// ---- P2POUs/BasicFunction/10_MES/CS_CodeTcp.TcPOU
FUNCTION_BLOCK PUBLIC CS_CodeTcp
VAR_INPUT
	bLON                           :BOOL; 	//  扫码开
	sRemoteHost: T_IPv4Addr; 			//扫码枪IP地址;
	bComOpen                  :BOOL; 	 //扫码Tcp 开
	binit_tcp:BOOL;							//功能块初始化，所有状态全部清零；
END_VAR

VAR_OUTPUT
	bComOpenDone          :BOOL;  //扫码Tcp 打开OK
    bCodeConError             :BOOL;//扫码通讯故障
	bDone                         :BOOL; //扫码完成
    bCodeError                  :BOOL;//扫码故障	
    strCode                       :STRING;//条码结果
	Code_State:INT;						//扫码结果 1：OK  2：NG
END_VAR

VAR_IN_OUT

END_VAR

VAR
	bLOFF                          :BOOL; 	//扫码关	
	bComClose                  :BOOL;  	//扫码Tcp 关
	fbTcpCon:FB_SocketConnect;
	fbTcpSend:FB_SocketSend;
	fbTcpRec:FB_SocketReceive;
	fbTcpClose: FB_SocketClose;
	bConnect: BOOL;//打开TCP连接;
	bClose: BOOL;		//关闭TCP连接;
	hTcpSock: T_HSOCKET;
	StrSend:STRING;
	StrReceive:STRING;
	StrReceive2:STRING:='';//clean;
	fbUdpCreate:FB_SocketUdpCreate;
	hUdp: T_HSOCKET;
	bCreate: BOOL;
	port: UDINT:=23;
	bSendTcp: BOOL;
	bReceiveTcp: BOOL;
	fbSwingHalt2: MC_Halt;
    TON01:TON;
	Lenth: UINT;
	StrSend2: STRING;
	bSendTcp2: BOOL;
	iComSetp: INT;
	bRectiveEN: BOOL;
	TON_3: Ton;
	TON_4: TON;
	tTon5: BOOL;
	TON_5: TON;
END_VAR




	Config();
	
	M_SendReceive();


	
	

	
	
	
	

	
	
	
	
	
	
	
	
	
	
	
	
	
	
	
	
	
(*	
   fbUdpCreate(
	sSrvNetId:= , 
	sLocalHost:= , 
	nLocalPort:= port, 
	bExecute:=bCreate , 
	tTimeout:= , 
	bBusy=> , 
	bError=> , 
	nErrId=> , 
	hSocket=> hUdp);
	
	
	*)

ACTION Config:
(*
功能块初始化；
外部给一个上升沿;
*)
TON_3(IN:=binit_tcp , PT:=T#2MS , Q=> , ET=> ); 
IF binit_tcp THEN
	iComSetp:=0;
	bComOpenDone:=FALSE;
    bCodeConError:=FALSE;
	bCodeError:=FALSE;
	bConnect:=FALSE;
	bClose :=TRUE;
	bDone:=FALSE;
    strCode:=StrReceive2;	 
	StrReceive:=StrReceive2;	 
	Code_State:=0;
	bRectiveEN:=FALSE;
	bSendTcp:=FALSE;
END_IF
IF TON_3.Q THEN
	binit_tcp:=FALSE;
	bClose :=FALSE;
END_IF

(*************************************************************)

IF bComOpen THEN
    bComOpenDone:=FALSE;
    bCodeConError:=FALSE;
    iComSetp:=100;
END_IF
  
 IF bComClose THEN
     bComOpenDone:=FALSE;
     bCodeConError:=FALSE;
     iComSetp:=200;
END_IF 
  

 CASE iComSetp OF 
   100:
	   bConnect:=TRUE;	
	   bClose:=FALSE;
	   bComOpen:=FALSE;
	   iComSetp:=110;
  110:
	  IF bConnect  THEN
		  bConnect:=FALSE;	
		   iComSetp:=120;
	  ELSIF fbTcpCon.bError THEN
		  iComSetp:=999;
	 END_IF
  120:
	 IF fbTcpCon.hSocket.handle>0  THEN
		bComOpenDone:=TRUE;//扫码枪连接成功；
		 iComSetp:=666;
	 ELSIF  NOT fbTcpCon.bBusy AND fbTcpCon.hSocket.handle=0  THEN
		iComSetp:=999;
	 END_IF

  200:
	   bConnect:=FALSE;	
	   bClose:=TRUE;
	   bComClose:=FALSE;
       iComSetp:=210;
  210:
	  IF fbTcpClose.bBusy THEN
		  bConnect:=FALSE;	
		   iComSetp:=666;
	 END_IF
  
  999:
	   bCodeConError:=TRUE;
	   iComSetp:=0;
END_CASE

fbTcpCon(
	sSrvNetId:= ''   ,                                     
	sRemoteHost:=sRemoteHost,     
	nRemotePort:= 23, 
	bExecute:=bConnect , 
	tTimeout:= , 
	bBusy=> , 
	bError=> , 
	nErrId=> , 
	hSocket=>hTcpSock );

fbTcpClose(
	sSrvNetId:= ''   , 
	hSocket:=hTcpSock , 
	bExecute:=bClose , 
	tTimeout:=T#5S , 
	bBusy=> , 
	bError=> , 
	nErrId=> );
END_ACTION

ACTION M_SendReceive:
(*
扫码失败返回“NG”；
 MEMSET(ADR(StrReceive2),0,SIZEOF(StrReceive2)); 
*)
TON_5(IN:=tTon5, PT:=T#4S , Q=> , ET=> ); 
IF TON_5.Q THEN
	tTon5:=FALSE;
END_IF

 IF bLON   AND  bComOpenDone   THEN
	StrReceive2:='$00$00$00$00$00$00$00$00$00$00$00$00$00$00$00$00$00$00$00$00$00$00$00$00$00$00$00$00$00$00$00$00';
	StrReceive:=StrReceive2;	 
	strCode:=StrReceive2;
	tTon5:=TRUE;
	IF StrReceive='' THEN
		 StrSend:='+';
		 bSendTcp:=TRUE;
		 bLON:=FALSE;
		 bDone:=FALSE;
		 bCodeError:=FALSE;
		 strCode:='';
		 Lenth:=SIZEOF(StrSend);
		 bRectiveEN:=TRUE;
	  END_IF
 END_IF
 

  IF bLOFF OR bCodeConError THEN
     StrSend:='+';
	 bSendTcp:=TRUE;
	 bLOFF:=FALSE;
	 bDone:=FALSE;
	 bCodeError:=FALSE;
	 strCode:='';
	 bComOpenDone:=FALSE;
	 iComSetp:=0;
	 Code_State:=0;
	 Lenth:=SIZEOF(StrSend2);
  END_IF

 //发送； 
fbTcpSend(
		sSrvNetId:= , 
		hSocket:=hTcpSock , 
		cbLen:=SIZEOF(StrSend), 
		pSrc:= ADR(StrSend), 
		bExecute:= bSendTcp, 
		tTimeout:= T#2S , 
		bBusy=> , 
		bError=> , 
		nErrId=> );
	
	IF TON01.Q THEN
		bSendTcp:=FALSE;
	END_IF

	
//接收;
bReceiveTcp:=tTon5 AND NOT bReceiveTcp AND  bRectiveEN     ;
fbTcpRec(
	sSrvNetId:= , 
	hSocket:= hTcpSock, 
	cbLen:=SIZEOF(StrReceive) , 
	pDest:=ADR(StrReceive) , 
	bExecute:=bReceiveTcp , 
	tTimeout:= T#5S, 
	bBusy=> , 
	bError=> , 
	nErrId=> , 
	nRecBytes=> );
	
(*接收数据超时；	*)

TON_4(IN:=bRectiveEN, PT:=T#4S , Q=> , ET=> ); 
IF TON_4.Q THEN
		IF(  StrReceive='' )OR ( LEN(STR:=StrReceive )<>2 AND LEN(STR:=StrReceive )<>15 )THEN	
				strCode:=StrReceive;
			   StrReceive:='';
			   bRectiveEN:=FALSE;
			   bCodeError:=TRUE;
			   Code_State:=2;			//拍照失败；
		END_IF
END_IF

(*数据位数不对报警*)
IF tTon5 AND LEN(STR:=StrReceive )<>0 AND LEN(STR:=StrReceive )<>2 AND LEN(STR:=StrReceive )<>15  THEN
				strCode:=StrReceive;
			   StrReceive:='';
			   bRectiveEN:=FALSE;
			   bCodeError:=TRUE;
			   Code_State:=2;			//拍照失败；
END_IF

(*截取数据判断；*)
IF StrReceive<>''THEN
		IF NOT bLON AND NOT fbTcpRec.bBusy THEN
			bRectiveEN:=FALSE;
			bSendTcp:=FALSE;
		END_IF

IF tTon5 AND LEN(STR:=StrReceive )>=2 AND LEN(STR:=StrReceive )<=15 AND FIND(STR1:=StrReceive , STR2:='ERROR' )=0 THEN
	  strCode:=StrReceive;
	  StrReceive:='';
     bRectiveEN:=FALSE;
	 bDone:=TRUE;
	 		IF strCode='NG' THEN
				Code_State:=2;//拍照失败；
			ELSE
				Code_State:=1;//拍照成功；
			END_IF
	END_IF  		
	ELSIF FIND(STR1:=StrReceive , STR2:='ERROR2222' )<>0  THEN 
	  strCode:=StrReceive;
	  StrReceive:='';
       bRectiveEN:=FALSE;
	  bCodeError:=TRUE;
	  Code_State:=2;//拍照失败；

END_IF


IF stSysState.hmiReset THEN
	bCodeConError:=FALSE;
	bCodeError:=FALSE;
END_IF
END_ACTION

END_FUNCTION_BLOCK

// ---- P2POUs/BasicFunction/03_Motion/CS_SetpMoter.TcPOU
FUNCTION_BLOCK CS_SetpMoter
VAR_INPUT
END_VAR
VAR_OUTPUT
END_VAR
VAR
	
	
END_VAR

VAR_IN_OUT
stSetpMotor:ST_SetpMotor;//电芯出料步进电机	
END_VAR
	

VAR
iSensorCount: INT;
//R_TRIG10:R_TRIG;
//F_TRIG10:F_TRIG;
R_trig20:R_TRIG;
R_trig21:R_TRIG;
R_trig23:R_TRIG;
R_trig22:R_TRIG;
TON50:TON;
TON51:TON;
TON52:TON;
TON53:TON;
TON54:TON;
iSetp3:INT;   //电芯转移流程


END_VAR

(*********************步进电机控制*****************************)
//步进点动
stSetpMotor.bo_Up:=stSetpMotor.bJog_Up AND NOT stSetpMotor.biUpSensor ; //步进点动上升   
stSetpMotor.bo_Down:=stSetpMotor.bJog_Down AND NOT stSetpMotor.biDownSensor ;   //步进点动下降   

//步进回原点
iSensorCount:=BOOL_TO_INT(stSetpMotor.biUpSensor)+ BOOL_TO_INT(stSetpMotor.biDownSensor);
R_trig20(CLK:=stSetpMotor.bHome , Q=> );
IF R_trig20.Q  AND iSensorCount<=1 THEN
   iSetp3:=88;
   stSetpMotor.bHome:=FALSE;
   stSetpMotor.HomeDone:=FALSE;
   stSetpMotor.bPoleFull:=FALSE;
END_IF

R_trig21(CLK:=stSetpMotor.bGoWorkPos , Q=> ); //GO工作位置  
IF R_trig21.Q  THEN  //AND iSensorCount<=1
   stSetpMotor.bJog_Down:=FALSE;
   stSetpMotor.bJog_Up:=FALSE;
   iSetp3:=99;	
   stSetpMotor.HomeDone:=FALSE;
   stSetpMotor.bGoWorkPos:=FALSE;
   stSetpMotor.WorkPosDone:=FALSE;
   stSetpMotor.bPoleFull:=FALSE;
END_IF

R_trig23(CLK:=stSetpMotor.bLeaveWorkPos , Q=> ); //离开工作位置  
IF R_trig23.Q  THEN  //AND iSensorCount<=1
   stSetpMotor.bJog_Down:=FALSE;
     stSetpMotor.bJog_Up:=FALSE;
    iSetp3:=97;	
	stSetpMotor.HomeDone:=FALSE;
   stSetpMotor.bLeaveWorkPos:=FALSE;
   stSetpMotor.WorkPosDone:=FALSE;
   stSetpMotor.bPoleFull:=FALSE;
END_IF

TON50(IN:= , PT:=T#20MS , Q=> , ET=> );  //感应原点后延时
TON51(IN:= , PT:=T#20MS , Q=> , ET=> );  //对射感应原点后延时
TON52(IN:= , PT:=T#10S , Q=> , ET=> );  //感应电芯报警
TON53(IN:= , PT:=T#300MS , Q=> , ET=> );  //感
TON54(IN:=iSetp3=200 , PT:=T#20S , Q=> , ET=> );  //回原超时
R_trig22(CLK:=iSensorCount=1 , Q=> );  

IF TON54.Q THEN
	//stSetpMotor.bError[1]:=TRUE;//回原超时
	stSetpMotor.bJog_Down:=FALSE;
	stSetpMotor.bJog_Up:=FALSE; 	
	iSetp3:=0;
END_IF

CASE iSetp3 OF   	
88:  
   IF stSetpMotor.biDownSensor THEN  //本来就在原点  回原完成
	   TON50.IN:=TRUE; 
	   TON52.IN:=FALSE;
	   IF TON50.Q THEN
		   stSetpMotor.HomeDone:=TRUE;
		   stSetpMotor.bJog_Down:=FALSE;
		   stSetpMotor.bJog_Up:=FALSE; 		   
		   TON50.IN:=FALSE;  
		   iSetp3:=666;   
	   END_IF
   //ELSIF  stSetpMotor.biDownSensor THEN  
	    // iSetp3:=100; 
   ELSIF  stSetpMotor.biUpSensor THEN 	   
	      iSetp3:=200;    
   ELSE                //没在任何感应 
       iSetp3:=200;    //默认往参考点回原点
   END_IF
 (* 
100:  //上升
	   stSetpMotor.bJog_Down:=FALSE;
	   stSetpMotor.bJog_Up:=TRUE;      //下限位 往上  碰到 mid2停
	    IF stSetpMotor.biRefSensor THEN
		  iSetp3:=88;	
		END_IF*)   
200:   //下降
	   stSetpMotor.bJog_Down:=TRUE;
	   stSetpMotor.bJog_Up:=FALSE; 
	   IF  R_trig22.Q THEN   //下将过程中碰到限位
		   iSetp3:=88;	 
	   END_IF   
  
(*************************对射位置***********************)   
99:    //在原位先上升    
	   stSetpMotor.bJog_Down:=FALSE;
	    stSetpMotor.bJog_Up:=TRUE;  
		TON52.IN:=TRUE;
		 iSetp3:=300;    	   
300: //对射检测
	 IF stSetpMotor.biUpSensor  THEN 
	    stSetpMotor.bJog_Down:=TRUE;
	    stSetpMotor.bJog_Up:=FALSE; 
	 END_IF

		IF stSetpMotor.biSensor   THEN //stSetpMotor.biSensor
		   TON51.IN:=TRUE; 
		   IF TON51.Q THEN 
			   stSetpMotor.WorkPosDone:=TRUE;
               stSetpMotor.bJog_Down:=FALSE;
			   stSetpMotor.bJog_Up:=FALSE; 
		       TON51.IN:=FALSE; 
			   iSetp3:=666;   
			END_IF   	
		END_IF
		
(**************************离开对射位置********************************)  		
97:     
     IF  NOT stSetpMotor.bJog_Down AND NOT stSetpMotor.bJog_Up   THEN //升降轴上升到位 
		 stSetpMotor.bJog_Down:=TRUE;
		 stSetpMotor.bJog_Up:=FALSE;
         TON53.IN:=TRUE;
		 iSetp3:=400; 
	 END_IF		
		
400:  //步进电机回原位
	     IF TON53.Q AND NOT stSetpMotor.biSensor THEN//stSetpMotor.biSensor
		   stSetpMotor.WorkPosDone:=TRUE;
		    stSetpMotor.bJog_Down:=FALSE;
		    stSetpMotor.bJog_Up:=FALSE;	 
		     TON53.IN:=FALSE;
		   iSetp3:=666; 
		 END_IF
	     IF stSetpMotor.biDownSensor  THEN
		     stSetpMotor.bJog_Down:=FALSE;
		      stSetpMotor.bJog_Up:=FALSE;	
             TON53.IN:=FALSE; 
		   // bAlarm:=TRUE;  
            stSetpMotor.bPoleFull:=TRUE;  
		    iSetp3:=666; 
		 END_IF							
END_CASE

END_FUNCTION_BLOCK

// ---- P2POUs/BasicFunction/12_User2/FB_AxisHandautomatic.TcPOU
FUNCTION_BLOCK FB_AxisHandautomatic
VAR_INPUT
    Notmoing:BOOL;//主轴停止中
	Run:BOOL;//自动
	i:INT;
	j: INT;
	Reset:BOOL;//手自动对比复位
END_VAR

VAR_OUTPUT
error :BOOL ;
END_VAR

VAR
	step:INT ;
	rRun : R_TRIG;
	fRun: F_TRIG;

	Pause_CMD:ARRAY[1..185] OF LREAL ; //手自动对比位置
	Handautomark:BOOL;//手自动对比标志
	K: INT;
	K1: INT;

END_VAR

VAR_IN_OUT

END_VAR




rRun(CLK:= Run , Q=> );
fRun(CLK:= Run , Q=> );


		IF fRun.Q THEN
			step:=100; 
		END_IF
		
	CASE step OF	
		100:
		   IF Notmoing THEN
			 step:=110;  
		   END_IF
	    110:    
	        Handautomark:=TRUE;
			FOR K:=i TO ((i+j)-1) DO 
			Pause_CMD[K]:=arrAxisCtrl[K].Status.fActPos;
			END_FOR
	        step:=120;    
	END_CASE
		

	   IF rRun.Q AND Handautomark THEN
				FOR K:=i TO ((i+j)-1) DO 
						IF  ABS(Pause_CMD[K]-arrAxisCtrl[K].Status.fActPos)>=0.2 THEN
						Axis_error[k]:=TRUE;
						END_IF
						
						IF Axis_error[k]   THEN
							error:=TRUE;
						END_IF
				END_FOR
				    Handautomark:=FALSE;
		END_IF
		
		IF stSysState.btnReset OR  stSysState.hmiReset  THEN
			   error:=FALSE;
			   FOR K1:=1 TO 185 DO 
				       Axis_error [K1]:=FALSE;
			   END_FOR
		END_IF
		
		IF Reset THEN
			 Handautomark:=FALSE;
		END_IF

END_FUNCTION_BLOCK

// ---- P2POUs/POUS/FingerprintKey.TcPOU
PROGRAM FingerprintKey
VAR
	MachineId: STRING(2);//叠台指纹编号对应标志
	ID: STRING(49);
	Level: STRING(49);
	LoginSuccess: BOOL;//指纹匹配成功
	Keyton:  ARRAY[0..10] OF TON;//1:获取用户及权限延时
	LevelHMI_Read: BYTE;//触摸屏权限，用于触摸屏读取用户索引
	PassWord: STRING(16);//触摸屏密码，用于触摸屏读取用户对应密码
	LevelHMI_Write: INT;//触摸屏权限，用于触摸屏反馈给PLC
	KeyStep: INT;//权限判断自动
	cheshi:BOOL;
	blogin: BOOL;
	blogout: BOOL;
	rKey:  ARRAY[0..10] OF R_TRIG;
	//error:ARRAY[0..60] OF BOOL;
END_VAR

Keyton[1](IN:=LoginSuccess,PT:=T#100MS , Q=> , ET=> );

IF GVL_Par.DT_FingerprintKey.MachineId='03' THEN
	IF GVL_Par.DT_FingerprintKey.Result='Success' THEN
		LoginSuccess:=TRUE;//指纹匹配成功
	END_IF	
END_IF

CASE KeyStep OF
0:
	IF Keyton[1].Q THEN
		IF GVL_Par.DT_FingerprintKey.UserId<>'' AND GVL_Par.DT_FingerprintKey.UserClassLevel<>'' THEN
			ID:=GVL_Par.DT_FingerprintKey.UserId;
			Level:=GVL_Par.DT_FingerprintKey.UserClassLevel;
			LevelHMI_Read:=0;
			LevelHMI_Write:=0;
			blogin:=FALSE;
			blogout:=FALSE;
			IF ID=GVL_Par.DT_FingerprintKey.UserId AND Level=GVL_Par.DT_FingerprintKey.UserClassLevel AND NOT blogin THEN
				GVL_Par.DT_FingerprintKey.Result:='';
				KeyStep:=100;
			END_IF
		END_IF
	END_IF
100://用户权限判断	(触摸屏读取时，采用用户索引，顺序要与触摸屏用户顺序一致）
	Keyton[1].IN:=FALSE;
	IF Level='PRD' THEN
		LevelHMI_Read:=1;
		//PassWord:='1111';
		IF LevelHMI_Read=1  THEN//AND PassWord='1111'
			KeyStep:=200;
		END_IF
	ELSIF Level='ME' THEN
		LevelHMI_Read:=2;
		//PassWord:='SWD123';
		IF LevelHMI_Read=2  THEN//AND PassWord='SWD123'
			KeyStep:=200;
		END_IF
	ELSIF Level='PRJ' THEN
		LevelHMI_Read:=3;
		//PassWord:='SWDQDJ';
		IF LevelHMI_Read=3  THEN//AND PassWord='SWDQDJ'
			KeyStep:=200;
		END_IF
	ELSIF Level='GYS' THEN
		LevelHMI_Read:=4;
		//PassWord:='YK556';
		IF LevelHMI_Read=4 THEN// AND PassWord='YK556'
			KeyStep:=200;
		END_IF
	ELSIF Level='QA' THEN
		LevelHMI_Read:=5;
		//PassWord:='OYX98766';
		IF LevelHMI_Read=5  THEN//AND PassWord='OYX98766'
			KeyStep:=200;
		END_IF
	ELSIF Level='KF' THEN
		LevelHMI_Read:=6;
		//PassWord:='0513';
		IF LevelHMI_Read=6  THEN//AND PassWord='0513'
			KeyStep:=200;
		END_IF
	ELSIF Level='Safe' THEN
		LevelHMI_Read:=7;
		//PassWord:='87558';
		IF LevelHMI_Read=7 THEN//AND PassWord='87558'
			KeyStep:=200;
		END_IF
	ELSE
		LoginSuccess:=FALSE;
		Level:='';
		GVL_Par.DT_FingerprintKey.Result:='';
		GVL_Par.DT_FingerprintKey.UserId:='';
		GVL_Par.DT_FingerprintKey.UserClassLevel:='';
		GVL_Par.DT_FingerprintKey.MachineId:='';
		blogin:=FALSE;
		blogout:=FALSE;
		KeyStep:=0;
		//error[1]:=TRUE;指纹未录入弹窗
	END_IF
200:
	blogin:=TRUE;
	LoginSuccess:=FALSE;
	KeyStep:=300;
300:
	IF LevelHMI_Write=1 THEN
		LevelHMI_Read:=0;
		PassWord:='';
		LoginSuccess:=FALSE;
		Level:='';
		GVL_Par.DT_FingerprintKey.Result:='';
		GVL_Par.DT_FingerprintKey.UserId:='';
		GVL_Par.DT_FingerprintKey.UserClassLevel:='';
		GVL_Par.DT_FingerprintKey.MachineId:='';
		blogin:=FALSE;
		blogout:=FALSE;
		KeyStep:=0;
	END_IF
END_CASE

END_PROGRAM

// ---- P3POUs/POUs/P3MAIN.TcPOU
PROGRAM P3MAIN
VAR
	fbDataXML  :FB_DataXMLP3;  
	bSave: BOOL;
	rt10: R_TRIG;
	bReadDataFirstCyle: BOOL;
	testii: INT;
	bSaveDataTest: BOOL;
	testii2: INT;
	bReadDataCyle2: BOOL;
	rtSaveData: R_TRIG;



	BUSY: BOOL;
	ERR: BOOL;
	ERRID: UDINT;
	CSData:    CS_Data;
	

	THNN: INT;
	MA100: BOOL;
	A1: BOOL;
	D1: BOOL;
	A2: BOOL;
	A3: BOOL;
	
	//iShort:        IShortTest;
	D2: INT;
	//stTime: TIMESTRUCT;
	strTime: STRING;
	BY1:  BYTE;
	AA1: BOOL;
	btest: BOOL;
	iPower: INT;
	iPowerSetp: INT;
	bytePower: BYTE:=16#01;
	boPower2: BOOL;
	k: INT:=1;
	PowerOnDone: BOOL;
   
	rt:ARRAY[1..5]OF R_TRIG;//上升沿触发
	tRead			:TON;
END_VAR

VAR
	bFirstCycle										        	:BOOL;	(*初始化用的*)
(*保存掉电保持参数*)
	//FB_WritePersistentData1								: FB_WritePersistentData;
	tCycleTimer											: TON;
	bWrite												: BOOL;    (*定时自动保存*)
(*系统重启*)
	tNtDelayReset										:TON;
	bReboot											: BOOL;	(*重启系统的变量*)
//	NT_Reboot1											: NT_Reboot;
(*系统关机*)
	//NT_Shutdown1										: NT_Shutdown;
	tNtDelayShutdown									: TON;
	bShutdown											: BOOL;
(*远程桌面接管*)
	OpenRemoteDesktop									: NT_StartProcess;
	timerHMI											:TON;
(*系统时间获取*)
//	NT_GetTime1											: NT_GetTime;
(*心跳信号*)
	bHeartBeat											:BOOL;
	tHeartBeatTime										:TIME:=t#0.5s;
	TonHeartBeat										:TON;

	TaskInfo											:	TaskInfoCtrl;
	loadParaStep: UINT;
	i: UINT;	

    tonPowerOn  :Tc2_Standard.TON;
    tonPower       :Tc2_Standard.TON;


     STR1: STRING:='20200412160000';
	 STR2: STRING:='12345678ABCDE';
	 STR3: STRING:='SSDDFF1234  JJJJ';
	 size:UDINT;
END_VAR

 VAR
     REST_TON :ARRAY[1..10] OF Tc2_Standard.TON;
END_VAR


P3IOLink();

IF tonPowerOn.ET>=T#5S THEN
    P3Main.RecipeData();
END_IF

tonPowerOn(IN:=PowerOnDone , PT:=T#15S , Q=> , ET=> );  //上电延时5S

IF tonPowerOn.Q AND fbDataXML.bReadParDone THEN
  P3MainState();  
ELSE
   Power();//接触器上电
END_IF




 
 

//冷压负极软限位写入
fADSWrite_Limit[1](
	IDXGRP_W:= 16#50C0, 
	IDXOFFS_W:= 16#D, 
	IDXOFFSLimit_W:= 16#B, 
	bSetButton:= HMI_SetButton[1], 
	bSetLimitButton:=P3User2_Par.HMI_Button[1] , 
	fSavePositionBias:=P3User2_Par.fSavePositionBias[1] , 
	AxisNo:=165 , 
	ADSMark:=ADSRefMark,
	bWriteAlarm=>HMI_ADSAlarm[1] ,
	fSaveBias=>HMI_SaveBias[1]);

//冷压正极软限位写入
fADSWrite_Limit[2](
	IDXGRP_W:= 16#50C0, 
	IDXOFFS_W:= 16#E, 
	IDXOFFSLimit_W:= 16#C, 
	bSetButton:= HMI_SetButton[2], 
	bSetLimitButton:=P3User2_Par.HMI_Button[2] , 
	fSavePositionBias:=P3User2_Par.fSavePositionBias[2] , 
	AxisNo:=165 , 
	ADSMark:=ADSRefMark,
	bWriteAlarm=>HMI_ADSAlarm[2] ,
	fSaveBias=>HMI_SaveBias[2]);
	
//热压负极软限位写入	
fADSWrite_Limit[3](
	IDXGRP_W:= 16#50C5, 
	IDXOFFS_W:= 16#D, 
	IDXOFFSLimit_W:= 16#B, 
	bSetButton:= HMI_SetButton[3], 
	bSetLimitButton:=P3User2_Par.HMI_Button[3] , 
	fSavePositionBias:=P3User2_Par.fSavePositionBias[3] , 
	AxisNo:=170 , 
	ADSMark:=ADSRefMark,
	bWriteAlarm=>HMI_ADSAlarm[3] ,
	fSaveBias=>HMI_SaveBias[3]);

	
//热压正极软限位写入
fADSWrite_Limit[4](
	IDXGRP_W:= 16#50C5, 
	IDXOFFS_W:= 16#E, 
	IDXOFFSLimit_W:= 16#C, 
	bSetButton:= HMI_SetButton[4], 
	bSetLimitButton:=P3User2_Par.HMI_Button[4] , 
	fSavePositionBias:=P3User2_Par.fSavePositionBias[4] , 
	AxisNo:=170 , 
	ADSMark:=ADSRefMark,
	bWriteAlarm=>HMI_ADSAlarm[4],
	fSaveBias=>HMI_SaveBias[4] );
	
	
 
 
 	
//1#贴胶进退负极软限位写入	
fADSWrite_Limit[5](
	IDXGRP_W:= 16#505B, 
	IDXOFFS_W:= 16#D, 
	IDXOFFSLimit_W:= 16#B, 
	bSetButton:= HMI_SetButton[5], 
	bSetLimitButton:=P3User2_Par.HMI_Button[5] , 
	fSavePositionBias:=P3User2_Par.fSavePositionBias[5] , 
	AxisNo:=43 , 
	ADSMark:=ADSRefMark,
	bWriteAlarm=>HMI_ADSAlarm[5] ,
	fSaveBias=>HMI_SaveBias[5]);

	
//1#贴胶进退正极软限位写入
fADSWrite_Limit[6](
	IDXGRP_W:= 16#505B, 
	IDXOFFS_W:= 16#E, 
	IDXOFFSLimit_W:= 16#C, 
	bSetButton:= HMI_SetButton[6], 
	bSetLimitButton:=P3User2_Par.HMI_Button[6] , 
	fSavePositionBias:=P3User2_Par.fSavePositionBias[6] , 
	AxisNo:=43 , 
	ADSMark:=ADSRefMark,
	bWriteAlarm=>HMI_ADSAlarm[6],
	fSaveBias=>HMI_SaveBias[6] );	
	

//2#贴胶进退负极软限位写入	
fADSWrite_Limit[7](
	IDXGRP_W:= 16#5089, 
	IDXOFFS_W:= 16#D, 
	IDXOFFSLimit_W:= 16#B, 
	bSetButton:= HMI_SetButton[7], 
	bSetLimitButton:=P3User2_Par.HMI_Button[7] , 
	fSavePositionBias:=P3User2_Par.fSavePositionBias[7] , 
	AxisNo:=89 , 
	ADSMark:=ADSRefMark,
	bWriteAlarm=>HMI_ADSAlarm[7] ,
	fSaveBias=>HMI_SaveBias[7]);

	
//2#贴胶进退正极软限位写入
fADSWrite_Limit[8](
	IDXGRP_W:= 16#5089, 
	IDXOFFS_W:= 16#E, 
	IDXOFFSLimit_W:= 16#C, 
	bSetButton:= HMI_SetButton[8], 
	bSetLimitButton:=P3User2_Par.HMI_Button[8] , 
	fSavePositionBias:=P3User2_Par.fSavePositionBias[8] , 
	AxisNo:=89 , 
	ADSMark:=ADSRefMark,
	bWriteAlarm=>HMI_ADSAlarm[8],
	fSaveBias=>HMI_SaveBias[8] );	
	
	
	
 //3#贴胶进退负极软限位写入	
fADSWrite_Limit[9](
	IDXGRP_W:= 16#50B7, 
	IDXOFFS_W:= 16#D, 
	IDXOFFSLimit_W:= 16#B, 
	bSetButton:= HMI_SetButton[9], 
	bSetLimitButton:=P3User2_Par.HMI_Button[9] , 
	fSavePositionBias:=P3User2_Par.fSavePositionBias[9] , 
	AxisNo:=135 , 
	ADSMark:=ADSRefMark,
	bWriteAlarm=>HMI_ADSAlarm[9] ,
	fSaveBias=>HMI_SaveBias[9]);

	
//3#贴胶进退正极软限位写入
fADSWrite_Limit[10](
	IDXGRP_W:= 16#50B7, 
	IDXOFFS_W:= 16#E, 
	IDXOFFSLimit_W:= 16#C, 
	bSetButton:= HMI_SetButton[10], 
	bSetLimitButton:=P3User2_Par.HMI_Button[10] , 
	fSavePositionBias:=P3User2_Par.fSavePositionBias[10] , 
	AxisNo:=135 , 
	ADSMark:=ADSRefMark,
	bWriteAlarm=>HMI_ADSAlarm[10],
	fSaveBias=>HMI_SaveBias[10] );
 
	
 
 
 //后段贴胶进退负极软限位写入	
fADSWrite_Limit[11](
	IDXGRP_W:= 16#50CD, 
	IDXOFFS_W:= 16#D, 
	IDXOFFSLimit_W:= 16#B, 
	bSetButton:= HMI_SetButton[11], 
	bSetLimitButton:=P3User2_Par.HMI_Button[11] , 
	fSavePositionBias:=P3User2_Par.fSavePositionBias[11] , 
	AxisNo:=178 , 
	ADSMark:=ADSRefMark,
	bWriteAlarm=>HMI_ADSAlarm[11] ,
	fSaveBias=>HMI_SaveBias[11]);

	
//后段贴胶进退正极软限位写入
fADSWrite_Limit[12](
	IDXGRP_W:= 16#50CD, 
	IDXOFFS_W:= 16#E, 
	IDXOFFSLimit_W:= 16#C, 
	bSetButton:= HMI_SetButton[12], 
	bSetLimitButton:=P3User2_Par.HMI_Button[12] , 
	fSavePositionBias:=P3User2_Par.fSavePositionBias[12] , 
	AxisNo:=178 , 
	ADSMark:=ADSRefMark,
	bWriteAlarm=>HMI_ADSAlarm[12],
	fSaveBias=>HMI_SaveBias[12] ); 
 
	 REST_TON[1](IN:=HMI_SetButton[6] , PT:=T#0.5S , Q=> , ET=>);
	 REST_TON[2](IN:=HMI_SetButton[8] , PT:=T#0.5S , Q=> , ET=>);
	 REST_TON[3](IN:=HMI_SetButton[10] , PT:=T#0.5S , Q=> , ET=>);
	 REST_TON[4](IN:=HMI_SetButton[12] , PT:=T#0.5S , Q=> , ET=>);

 IF  REST_TON[1].Q THEN
	 HMI_SetButton[6]:=FALSE;
END_IF 

 IF  REST_TON[2].Q THEN
	 HMI_SetButton[8]:=FALSE;
END_IF 

 IF  REST_TON[3].Q THEN
	 HMI_SetButton[10]:=FALSE;
END_IF 

 IF  REST_TON[4].Q THEN
	 HMI_SetButton[12]:=FALSE;
END_IF 

 IF  P2M1_MachCtrl.TJ_b.Stick_Judge THEN
	 P3User2_Par.fSavePositionBias[6]:= arrAxisPar[P2AxisNo.P2M1_GluingRetracting].arrTargetPoint[2]+2;
	 HMI_SetButton[6]:=TRUE;
ELSE 	 
	 P3User2_Par.fSavePositionBias[6]:= arrAxisPar[P2AxisNo.P2M1_GluingRetracting].arrTargetPoint[4]+2;
	 HMI_SetButton[6]:=TRUE;	 
 END_IF
 
 
  IF  P2M2_MachCtrl.TJ_b.Stick_Judge THEN
	 P3User2_Par.fSavePositionBias[8]:= arrAxisPar[P2AxisNo.P2M2_GluingRetracting].arrTargetPoint[2]+2;
	 HMI_SetButton[8]:=TRUE;
ELSE 	 
	 P3User2_Par.fSavePositionBias[8]:= arrAxisPar[P2AxisNo.P2M2_GluingRetracting].arrTargetPoint[4]+2;
	 HMI_SetButton[8]:=TRUE;	 
 END_IF
 
 
  IF  P2M3_MachCtrl.TJ_b.Stick_Judge THEN
	 P3User2_Par.fSavePositionBias[10]:= arrAxisPar[P2AxisNo.P2M3_GluingRetracting].arrTargetPoint[2]+2;
	 HMI_SetButton[10]:=TRUE;
ELSE 	 
	 P3User2_Par.fSavePositionBias[10]:= arrAxisPar[P2AxisNo.P2M3_GluingRetracting].arrTargetPoint[4]+2;
	 HMI_SetButton[10]:=TRUE;	 
 END_IF
 
 IF Step38=530 THEN
     P3User2_Par.fSavePositionBias[12]:=arrAxisPar[P3AxisNo.P3_TapeAdvance].arrTargetPoint[3]+2;
	 HMI_SetButton[12]:=TRUE;
 ELSIF Step38=535 THEN
      P3User2_Par.fSavePositionBias[12]:=arrAxisPar[P3AxisNo.P3_TapeAdvance].arrTargetPoint[5]+2;
	  HMI_SetButton[12]:=TRUE;
 END_IF

ACTION Power:
(***系统延时启动***)

tonPower(IN:= , PT:=T#1.5S , Q=> , ET=> );

CASE iPowerSetp OF
0:
    tonPower.IN:=TRUE;
    iPowerSetp:=10;
10:
   IF   tonPower.Q  THEN
      bytePower:=SHL(bytePower,1);
     
      tonPower(IN:=FALSE );
      k:=k+1;
     iPowerSetp:=20;
  END_IF
20:
    bytePower.0:=1;
    tonPower.IN:=TRUE;
    iPowerSetp:=30;
30:
   IF  k>=8 THEN
        iPowerSetp:=666;
       // bytePower:=16#00;
        PowerOnDone:=TRUE;
		ADSRefMark:=TRUE;//ADS写入标志
   ELSE
      iPowerSetp:=10;
   END_IF

END_CASE
 
bytePower.0;
bytePower.1;
bytePower.2;
bytePower.3;
bytePower.4;
bytePower.5;
bytePower.6;
bytePower.7;
END_ACTION

ACTION RecipeData:
IF NOT  bReadDataFirstCyle THEN //testii:=testii+1
	//fbDataXML.bRead:=NOT bDataValid;
	bReadDataFirstCyle:=TRUE;
END_IF


IF fbDataXML.bReadParDone AND bReadDataFirstCyle AND NOT  bReadDataCyle2 THEN   //  先备份数据暂时不开放 
	bReadDataCyle2:=TRUE;
END_IF

tCycleTimer(IN:=NOT tCycleTimer.Q , PT:=T#5M , Q=> , ET=> );
rtSaveData(CLK:=stHmiSysCmd.bSaveData , Q=> );
IF  rtSaveData.Q THEN
	bSaveDataTest:=TRUE;
END_IF
IF  tCycleTimer.Q   OR   bSaveDataTest THEN
    bSaveDataTest:=FALSE;
	fbDataXML.bSave:=TRUE;
	testii2:=testii2+1;
END_IF

rt[4](CLK:=stHmiSysCmd.bReadData (*AND P3_SystemRUN.iMode=3*) , Q=> );
rt[5](CLK:=PowerOnDone , Q=> );
tRead(IN:=PowerOnDone, PT:=T#3S , Q=> , ET=> );
IF   tRead.Q AND NOT fbDataXML.bReadParDone THEN
	 P3_Error[90]	:=TRUE;//上电后热压参数读取失败，请手动点读取参数
END_IF

fbDataXML(bSave:=fbDataXML.bSave AND NOT P3_Error[90] , bRead:=fbDataXML.bRead OR rt[4].Q OR rt[5].Q, bSaveParDone=> , bReadParDone=> );

fbDataXML.bSaveParDone;
fbDataXML.bReadParDone;




(*
tCycleTimer(IN:=NOT tCycleTimer.Q , PT:=T#333S , Q=>bSave , ET=> );
rt10(clk:=bSave);
IF NOT  bReadDataFirstCyle THEN //testii:=testii+1
	 fbDataXML.bRead:=TRUE;
	 testii:=testii+1;
	 bReadDataFirstCyle:=TRUE;
END_IF


IF fbDataXML.bReadParDone AND bReadDataFirstCyle AND NOT  bReadDataCyle2 THEN   //  先备份数据暂时不开放 
	
      fSavePositionBias:=P3User2_Par.fSavePositionBias   ;   
      HMI_Button:=P3User2_Par.HMI_Button   ;   

      Shield:=P3User2_Par.Shield;   
      Oven_Shield:=P3User2_Par.Oven_Shield;  
      LateBlanking_motor:=P3User2_Par.LateBlanking_motor;  
      Cold_par:=P3User2_Par.Cold_par;  	  
      Hot_par:=P3User2_Par.Hot_par;  		  
      Oven_finish:=P3User2_Par.Oven_finish;  
      Oven_Finish_Time:=P3User2_Par.Oven_Finish_Time;  
      Oven_cell:=P3User2_Par.Oven_cell;  
	  
      V:=P3User2_Par.V;  	  
      W:=P3User2_Par.W;  	
      B_OVEN:=P3User2_Par.B_OVEN;  
      Thick_Par:=P3User2_Par.Thick_Par;  
      Thick_MN:=P3User2_Par.Thick_MN;  
      Thick_Cell_Par:=P3User2_Par.Thick_Cell_Par;  	  
	  
      Door_Forbidden:=P3User2_Par.Door_Forbidden;  	
      Scan_IP:=P3User2_Par.Scan_IP;  
      Cold_Position:=P3User2_Par.Cold_Position;  
	  
      Thick_min:=P3User2_Par.Thick_min;  
      Thick_max:=P3User2_Par.Thick_max;  	  
      Oven_Time_S:=P3User2_Par.Oven_Time_S;  	
      Bounce_time:=P3User2_Par.Bounce_time;  
      Status_switching_time:=P3User2_Par.Status_switching_time;  
	  Standby_time:=P3User2_Par.Standby_time;    
	  
	
      bReadDataCyle2:=TRUE;
END_IF

rtSaveData(CLK:=stHmiSysCmd.bSaveData , Q=> );
IF  rtSaveData.Q THEN
	bSaveDataTest:=TRUE;
END_IF

IF  rt10.Q   OR   bSaveDataTest THEN
     P3User2_Par.fSavePositionBias:=fSavePositionBias; 	
      P3User2_Par.HMI_Button:=HMI_Button; 	

	P3User2_Par.Shield:=Shield; 	
	P3User2_Par.Oven_Shield:=Oven_Shield; 	
	P3User2_Par.LateBlanking_motor:=LateBlanking_motor; 	
	P3User2_Par.Cold_par:=Cold_par; 	
	P3User2_Par.Hot_par:=Hot_par; 	
	P3User2_Par.Oven_finish:=Oven_finish; 	
	P3User2_Par.Oven_Finish_Time:=Oven_Finish_Time; 	
	P3User2_Par.Oven_cell:=Oven_cell; 	
	
	
	P3User2_Par.V:=V; 	
	P3User2_Par.W:=W; 		
	P3User2_Par.B_OVEN:=B_OVEN; 	
	P3User2_Par.Thick_Par:=Thick_Par; 	
	P3User2_Par.Thick_MN:=Thick_MN; 		
	P3User2_Par.Thick_Cell_Par:=Thick_Cell_Par; 	
	
	P3User2_Par.Door_Forbidden:=Door_Forbidden; 	
	P3User2_Par.Scan_IP:=Scan_IP; 	
	P3User2_Par.Cold_Position:=Cold_Position; 	
	
	P3User2_Par.Thick_min:=Thick_min; 	
	P3User2_Par.Thick_max:=Thick_max; 		
	P3User2_Par.Oven_Time_S:=Oven_Time_S; 	
	P3User2_Par.Bounce_time:=Bounce_time; 	
	P3User2_Par.Status_switching_time:=Status_switching_time; 		
	P3User2_Par.Standby_time:=Standby_time; 	

    bSaveDataTest:=FALSE;
	fbDataXML.bSave:=TRUE;
	testii2:=testii2+1;
END_IF


fbDataXML(bSave:=fbDataXML.bSave AND P2SaveParDone,
                      bRead:=fbDataXML.bRead  AND P2ReadParDone, 
                      bSaveParDone=> , 
                      bReadParDone=>,
                      bError  =>                                          );

IF fbDataXML.bError THEN				  
P3_Error[92]:=TRUE;	
END_IF				  
D_Sys.P3SaveParDone:=fbDataXML.bSaveParDone;
D_Sys.P3ReadParDone:=fbDataXML.bReadParDone;
*)
END_ACTION

END_PROGRAM

// ---- P3POUs/P3FB/FB_DataXMLP3.TcPOU
FUNCTION_BLOCK FB_DataXMLP3
VAR_INPUT
    	bSave:BOOL;
	    bRead:BOOL;
		bReadSel:BOOL;//参数读取选择，TRUE=选择恢复上电备份的参数
END_VAR
VAR_OUTPUT
    	bSaveParDone      :BOOL;
	    bReadParDone     :BOOL;
END_VAR

VAR
	iDataSetp: INT;
	i1: INT;
	i2:BYTE;
	rt100:Tc2_Standard.R_TRIG;
	rt101:Tc2_Standard.R_TRIG;
	rt102:Tc2_Standard.R_TRIG;
	rt103:Tc2_Standard.R_TRIG;
	bSaveTemp: BOOL;
	bReadTemp: BOOL;
	sFilePath:STRING;//文件路径
	sNewFilePath:STRING;//新文件路径
	sOldFilePath:STRING;//旧文件路径
	sFileName:STRING;//文件名称
	sVarName:STRING;//变量名称
	fbXmlSrvRead				: FB_XmlSrvReadByName;//读取XML文件	
	fbXmlSrvWrite				: FB_XmlSrvWriteByName;//写入XML文件
	bFirstCycleFlg:BOOL;//首次执行标志位
	fbGetFileList: FB_GetFileList;//获取文件列表功能块
	stFindFileEntry:ARRAY[1..50] OF ST_FindFileEntry;//文件列表存放结构体	
	nFileBakStep:UINT;//文件备份步序
	fbFileDelete	: FB_FileDelete;//删除文件
	fbFileRename	: FB_FileRename;//文件重命名
	fbCreateDirectory:FB_CreateDirectory;//文件夹创建
END_VAR

M_WriteOrRead();
A_FileBak();

ACTION A_FileBak:
CASE nFileBakStep OF
	200:
		fbGetFileList(bExecute:=FALSE);
		fbFileDelete(bExecute:=FALSE);
		fbFileRename(bExecute:=FALSE);
		fbCreateDirectory(bExecute:=FALSE);
		nFileBakStep:=300;
	300:(*获取文件列表*)
		fbGetFileList.pFindFileListADR:=ADR(stFindFileEntry);
		fbGetFileList.u32FindFileListSizeOf:=SIZEOF(stFindFileEntry);
		fbGetFileList(bExecute:=TRUE,sgPathName:=sOldFilePath,sgFileType:='xml');	
		IF fbGetFileList.bDone THEN
			fbGetFileList(bExecute:=FALSE);
			nFileBakStep:=310;
		ELSIF fbGetFileList.bError THEN
			fbGetFileList(bExecute:=FALSE);
			nFileBakStep:=997;
		END_IF
	310:(*判断文件是否存在，文件存在则备份一次，文件不存在直接给完成信号*)
		FOR i2:=1 TO 50 DO
			IF stFindFileEntry[i2].sFileName=sFileName THEN//
				EXIT;
			END_IF
		END_FOR
		IF i2>50 THEN
			nFileBakStep:=666;
		ELSE
			nFileBakStep:=320;
		END_IF
	320:(*文件夹创建*)//后续更新后删除
	fbCreateDirectory(bExecute:=TRUE , sgPathName:=sNewFilePath, tTimeout:=T#1S );
	IF fbCreateDirectory.bDone THEN
		fbCreateDirectory(bExecute:=FALSE);
		nFileBakStep:=350;
	ELSIF fbCreateDirectory.bError THEN
		fbCreateDirectory(bExecute:=FALSE);
		nFileBakStep:=998;
	END_IF
	350:(*删除旧文件*)
		fbFileDelete.sPathName:= CONCAT(sNewFilePath,sFileName);
		fbFileDelete(bExecute:=TRUE,ePath:= PATH_GENERIC,tTimeout:=T#5S);
		IF NOT fbFileDelete.bBusy THEN
			fbFileDelete(bExecute:=FALSE);
			nFileBakStep:=360;
		END_IF
	360:(*重命名文件*)
		fbFileRename.sOldName:= CONCAT(sOldFilePath,sFileName);
		fbFileRename.sNewName:= CONCAT(sNewFilePath,sFileName);
		fbFileRename(bExecute:=TRUE,ePath:= PATH_GENERIC,tTimeout:=T#5S);
		IF NOT fbFileRename.bBusy THEN
			fbFileRename(bExecute:=FALSE);
			IF NOT fbFileRename.bError THEN
				nFileBakStep:=666;
			ELSE
				nFileBakStep:=999;
			END_IF			
		END_IF
END_CASE
END_ACTION

ACTION M_WriteOrRead:
rt100(CLK:=bSave , Q=> );//保存参数
rt101(CLK:=bRead , Q=> );//读取参数
IF rt100.Q THEN  //保存参数
    bSaveTemp:=TRUE;
	bReadTemp:=FALSE;
	bSaveParDone:=FALSE;
	iDataSetp:=50;
END_IF
IF rt101.Q THEN  //读取参数
    bReadTemp:=TRUE;
    bSaveTemp:=FALSE;
	bReadParDone:=FALSE;
	iDataSetp:=50;
END_IF

//rt102(CLK:=NOT bFirstCycleFlg AND NOT bReadTemp, Q=> );//首次上电自动备份参数
IF rt102.Q THEN  //首次上电自动备份参数
	iDataSetp:=50;
END_IF

CASE  iDataSetp OF 
	50:
		I1:=1;
		fbXmlSrvRead(bExecute:=FALSE);
		fbXmlSrvWrite(bExecute:=FALSE);
		bSave:=FALSE;
		bRead:=FALSE;
		iDataSetp:=100;
	 100:
	 	sFilePath:='C:\P3XML\';//保存文件路径
		CASE i1 OF 
			 1://轴参数
				sFileName:= 'P3arrAxisParV2.xml';
				sVarName:='P3Motion.arrAxisParV2';
			 2://arrTempPar
				sFileName  := 'P3arrTempPar.xml';
				sVarName:='P3Temperature.arrTempPar';
			3://P3par
				sFileName  := 'P3par.xml';
				sVarName:='P3Par.P3par';
			4://P3Data
				sFileName  := 'P3Data.xml';
				sVarName:='P3Par.P3User2_Par';
		END_CASE		
		
		IF  bSaveTemp THEN
			iDataSetp:=200;
		ELSIF  bReadTemp THEN
			iDataSetp:=300;
	//	ELSIF NOT bFirstCycleFlg THEN
	//		iDataSetp:=400;
		END_IF
		
	(********************保存数据流程：先备份原来参数再保存新参数，如果保存失败恢复至备份参数********************)
	200:(*开始备份*)
		sNewFilePath:=CONCAT(sFilePath,'Tmp\');
		sOldFilePath:=sFilePath;
		nFileBakStep:=200;//调用A_FileBak()进行文件备份
		iDataSetp:=210;
	210:(*文件备份状态判断*)
		IF nFileBakStep=666 THEN//文件备份成功，保存新参数
			iDataSetp:=230;
		ELSIF nFileBakStep>990 THEN//文件备份失败
			iDataSetp:=997;			
		END_IF
	230:(*保存新参数*)	
		fbXmlSrvWrite(
			bExecute:= TRUE, 
			ePath:=PATH_GENERIC , 
			nMode:=XMLSRV_ADDMISSING , 
			sSymName:=sVarName , 
			sFilePath:= CONCAT(sFilePath,sFileName), 
			sXPath:= '/DataEntry/Value', 
			tTimeout:= T#2S);
		IF NOT fbXmlSrvWrite.bBusy THEN
			fbXmlSrvWrite(bExecute:=FALSE);
			IF NOT fbXmlSrvWrite.bError THEN(*保存新参数成功*)
				iDataSetp:=500;
			ELSE(*保存新参数失败，恢复未写入新参数前的备份*)
				iDataSetp:=250;
			END_IF	
		END_IF
	250:(*保存新参数失败，恢复未写入新参数前的备份*)
		sOldFilePath:=CONCAT('Tmp\' ,sFileName);
		sNewFilePath:=sFilePath;
		nFileBakStep:=200;//调用A_FileBak()进行文件备份
		iDataSetp:=260;
	260:(*恢复文件状态判断*)
		IF nFileBakStep=666 THEN//文件恢复成功
			iDataSetp:=500;
		ELSIF nFileBakStep>990 THEN//文件恢复失败
			iDataSetp:=998;			
		END_IF		

	(********************参数读取流程********************)	
	300:(*参数读取选择，TRUE=选择恢复上电备份的参数*)
		IF bReadSel THEN
			sFilePath:=CONCAT(sFilePath,'Bak\');
		END_IF
		iDataSetp:=310;
	310:(*读取参数*)
		fbXmlSrvRead(
			bExecute:= TRUE, 
			ePath:=PATH_GENERIC , 
			nMode:=XMLSRV_ADDMISSING , 
			sSymName:= sVarName, 
			sFilePath:=CONCAT(sFilePath,sFileName) , 
			sXPath:='/DataEntry/Value' , 
			tTimeout:=T#2S);
		IF NOT fbXmlSrvRead.bBusy THEN
			fbXmlSrvRead(bExecute:=FALSE);
			IF NOT fbXmlSrvRead.bError THEN
				iDataSetp:=500;//读取成功
			ELSE
				iDataSetp:=999;//读取失败
			END_IF
		END_IF
		
	(********************上电自动备份流程，防止被覆盖********************)	
	400:
		sOldFilePath:=sFilePath;
		sNewFilePath:=CONCAT(sFilePath,'Bak\' );
		nFileBakStep:=200;//调用A_FileBak()进行文件备份
		iDataSetp:=410;
	410:
		IF nFileBakStep=666 THEN
				iDataSetp:=500;
		ELSIF nFileBakStep>990 THEN
				iDataSetp:=999;			
		END_IF
	500:(*继续写下个文件*)
		IF i1>=1 AND i1<4 THEN
			i1:=i1+1; 
			iDataSetp:=100; 
		ELSIF i1>=4 THEN
			IF  bSaveTemp THEN		
				bSaveParDone:=TRUE;
			ELSIF  bReadTemp THEN
				bReadParDone:=TRUE;
			ELSIF NOT bFirstCycleFlg THEN
				bFirstCycleFlg:=TRUE;
			END_IF
			bReadSel:=FALSE;
			bReadTemp:=FALSE;
			bSaveTemp:=FALSE;
			iDataSetp:=666;   
		END_IF
END_CASE
END_ACTION

END_FUNCTION_BLOCK

// ---- P3POUs/POUs/P3IOLink.TcPOU
PROGRAM P3IOLink
VAR
//	tFlash: TON;
//	bFlash:BOOL;
//	bIOinit: BOOL;
	XXX: INT;
	Q20815: BOOL;
	AA: INT;

     arrFilter_AD               : ARRAY[1..MaxAINo]  OF  FB_Filter_AD ;




	I1: INT;

    rt01   :Tc2_Standard.R_TRIG;
    rt02   :Tc2_Standard.R_TRIG;

     parDAOld                   :ARRAY[1..44] OF INT;   
END_VAR



P3_AI();
P3_AO();
P3_AutoLink();
P3_InPut();
P3_LimitSwitch();
P3_OutPut();

ACTION P3_AI:
//尾段下料

arrFilter_AD[28].AD	:=AI60[0];  //冷压压力检测
arrFilter_AD[29].AD	:=AI60[1];  //热压压力检测

//转换
FOR  I1:=28 TO 29   DO
  arrFilter_AD[I1](
	  iMode:=         2, 
	  AD:=					arrFilter_AD[I1].AD               , 
	  iLimitH:=         parFilterAD[I1].iLimitH  , 
	  iLimitL:=          parFilterAD[I1].iLimitL   , 
	  fRangeH:=      parFilterAD[I1].fRangeH , 
	  fRangeL:=       parFilterAD[I1].fRangeL , 
	  fPointNum:=   15 , 
	  Out_Value=>);
END_FOR

//P3Par.P3_AD_Press[1]:=arrFilter_AD[28].Out_Value;
//P3Par.P3_AD_Press[2]:=arrFilter_AD[29].Out_Value;
END_ACTION

ACTION P3_AO:

END_ACTION

ACTION P3_AutoLink:
//气缸映射
P3_Oven[1]:=P3CYNo.P3Oven1;
P3_Oven[2]:=P3CYNo.P3Oven2;
P3_Oven[3]:=P3CYNo.P3Oven3;
P3_Oven[4]:=P3CYNo.P3Oven4;
P3_Oven[5]:=P3CYNo.P3Oven5;
P3_Oven[6]:=P3CYNo.P3Oven6;
P3_Oven[7]:=P3CYNo.P3Oven7;
P3_Oven[8]:=P3CYNo.P3Oven8;
P3_Oven[9]:=P3CYNo.P3Oven9;
P3_Oven[10]:=P3CYNo.P3Oven10;
P3_Oven[11]:=P3CYNo.P3Oven11;
P3_Oven[12]:=P3CYNo.P3Oven12;
P3_Oven[13]:=P3CYNo.P3Oven13;
P3_Oven[14]:=P3CYNo.P3Oven14;
P3_Oven[15]:=P3CYNo.P3Oven15;
P3_Oven[16]:=P3CYNo.P3Oven16;
P3_Oven[17]:=P3CYNo.P3Oven17;
P3_Oven[18]:=P3CYNo.P3Oven18;
P3_Oven[19]:=P3CYNo.P3Oven19;
P3_Oven[20]:=P3CYNo.P3Oven20;
P3_Oven[21]:=P3CYNo.P3Oven21;




//力矩
	Torque_P3.ColdpreLineTorSet:=HMI_TorErrLimt_D[160];//冷呀上料夹平移报警力矩设定
	Torque_P3.ColdpreRetractTorSet:=HMI_TorErrLimt_D[161];//冷压上料夹进退报警力矩设定
	Torque_P3.ColdpreWhirlTorSet:=HMI_TorErrLimt_D[162];//冷压上料夹旋转报警力矩设定
	Torque_P3.ColdpreActTorSet:=HMI_TorErrLimt_D[165];//冷压驱动报警力矩设定
	Torque_P3.OvenCarryTorSet:=HMI_TorErrLimt_D[166];//烤箱上料夹搬运报警力矩设定
	Torque_P3.OvenRetractTorSet:=HMI_TorErrLimt_D[167];//烤箱上料夹进退报警力矩设定
	Torque_P3.HotpreActTorSet:=HMI_TorErrLimt_D[170];//热压驱动报警力矩设定
	Torque_P3.WeighLineTorSet:=HMI_TorErrLimt_D[171];//称重上料夹平移报警力矩设定
	Torque_P3.WeighWhirlTorSet:=HMI_TorErrLimt_D[173];//称重上料夹旋转报警力矩设定
	Torque_P3.SortingCarryTorSet:=HMI_TorErrLimt_D[174];//电芯分选夹搬运报警力矩设定
	Torque_P3.OffloadCarryTorSet:=HMI_TorErrLimt_D[176];//电芯下料夹搬运报警力矩设定
	
	Torque_P3.TapeTranslationTorSet:=HMI_TorErrLimt_D[178];//后段贴胶头进退报警力矩设定
	Torque_P3.TapeAdvanceTorSet:=HMI_TorErrLimt_D[179];//后段贴胶平移报警力矩设定
	
	Torque_P3.ColdpreLineTor:=iActTorque_D[160];//冷呀上料夹平移实时力矩
	Torque_P3.ColdpreRetractTor:=iActTorque_D[161];//冷压上料夹进退实时力矩
	Torque_P3.ColdpreWhirlTor:=iActTorque_D[162];//冷压上料夹旋转实时力矩
	Torque_P3.ColdpreActTor:=iActTorque_D[165];//冷压驱动实时力矩
	Torque_P3.OvenCarryTor:=iActTorque_D[166];//烤箱上料夹搬运实时力矩
	Torque_P3.OvenRetractTor:=iActTorque_D[167];//烤箱上料夹进退实时力矩
	Torque_P3.HotpreActTor:=iActTorque_D[170];//热压驱动实时力矩
	Torque_P3.WeighLineTor:=iActTorque_D[171];//称重上料夹平移实时力矩
	Torque_P3.WeighWhirlTor:=iActTorque_D[173];//称重上料夹旋转实时力矩
	Torque_P3.SortingCarryTor:=iActTorque_D[174];//电芯分选夹搬运实时力矩
	Torque_P3.OffloadCarryTor:=iActTorque_D[176];//电芯下料夹搬运实时力矩
	
	Torque_P3.TapeTranslationTor:=iActTorque_D[178];//后段贴胶头进退实时力矩
	Torque_P3.TapeAdvanceTor:=iActTorque_D[179];//后段贴胶平移实时力矩
	
(*
	HMI_TorAlarm_D[160]:=Torque_P3.ColdpreLineTorAlarm;//冷呀上料夹平移力矩超限报警
	HMI_TorAlarm_D[161]:=Torque_P3.ColdpreRetractTorAlarm;//冷压上料夹进退力矩超限报警
	HMI_TorAlarm_D[162]:=Torque_P3.ColdpreWhirlTorAlarm;//冷压上料夹旋转力矩超限报警
	HMI_TorAlarm_D[165]:=Torque_P3.ColdpreActTorAlarm;//冷压驱动力矩超限报警
	HMI_TorAlarm_D[166]:=Torque_P3.OvenCarryTorAlarm;//烤箱上料夹搬运力矩超限报警
	HMI_TorAlarm_D[167]:=Torque_P3.OvenRetractTorAlarm;//烤箱上料夹进退力矩超限报警
	HMI_TorAlarm_D[170]:=Torque_P3.HotpreActTorAlarm;//热压驱动力矩超限报警
	HMI_TorAlarm_D[171]:=Torque_P3.WeighLineTorAlarm;//称重上料夹平移力矩超限报警
	HMI_TorAlarm_D[173]:=Torque_P3.WeighWhirlTorAlarm;//称重上料夹旋转力矩超限报警
	HMI_TorAlarm_D[174]:=Torque_P3.SortingCarryTorAlarm;//电芯分选夹搬运力矩超限报警
	HMI_TorAlarm_D[176]:=Torque_P3.OffloadCarryTorAlarm;//电芯下料夹搬运力矩超限报警
*)	
	
	HMI_TorAlarm_D[178]:=Torque_P3.TapeTranslationTorSetAlarm;//后段贴胶头进退力矩超限报警
	HMI_TorAlarm_D[179]:=Torque_P3.TapeAdvanceTorSetAlarm;//后段贴胶平移力矩超限报警
END_ACTION

ACTION P3_InPut:
//尾段下料
//I601
arrCyCtrl[P3CYNo.P3ColdPressTensed].Io.DIOnSwitch:=I601[1]	;//	冷压麦拉张紧气缸伸出位
arrCyCtrl[P3CYNo.P3ColdPressTensed].Io.DIOFFSwitch:=I601[2]	;//	冷压麦拉张紧气缸缩回位
P3Senser.P3_ColdEmptyPress:=I601[3]	;//	冷压防空压感应
P3Senser.P3_ColdScapegoat :=I601[4]	;//	冷压替罪羊检测
arrCyCtrl[P3CYNo.P3OvenMoveClip].Io.DIONSwitch:=I601[5]	;//	烤箱上料夹张开位
arrCyCtrl[P3CYNo.P3OvenMoveClip].Io.DIOFFSwitch:=I601[6]	;//	烤箱上料夹闭合位

//P3Senser.P3_CacheSensor:=I601[7]	;//贴胶平台有料感应
P3Senser.P3_Securitydoorswitch13:=I601[7]	;//外罩门禁13

P3Senser.P3_Fxjgy:=I601[8]	;//	//分选夹电芯有无
P3Senser.P3_ShortTest_UpperFall:=I601[9]	;//	短路测试结果超上限
P3Senser.P3_ShortTest_LowerFall:=I601[10]   ;//	短路测试结果超下限
P3Senser.P3_ShortTest_Testing:=I601[11]     ;//	短路测试中
P3Senser.P3_ShortTest_Pass:=I601[12]        ;//	短路测试OK
P3Senser.P3_Czslgy:=I601[13];//称重上料夹电芯有无	
P3Senser.P3_Kxslgy:=I601[14];//烤箱上料夹电芯有无
P3Senser.P3_InLayOffPer1:=I601[15];//	下料位1允许放料
P3Senser.P3_InLayOffPer2:=I601[16];//	下料位2允许放料		
		
//I602		
arrCyCtrl[P3CYNo.P3Oven1].Io.DIOFFSwitch:=I602[1]	;//	1_1烤箱门关闭
arrCyCtrl[P3CYNo.P3Oven1].Io.DIONSwitch:=I602[2]	;//	1_1烤箱门打开
arrCyCtrl[P3CYNo.P3Oven4].Io.DIOFFSwitch:=I602[3]	;//	1_2烤箱门关闭
arrCyCtrl[P3CYNo.P3Oven4].Io.DIONSwitch:=I602[4]	;//	1_2烤箱门打开
arrCyCtrl[P3CYNo.P3Oven7].Io.DIOFFSwitch:=I602[5]	;//	1_3烤箱门关闭
arrCyCtrl[P3CYNo.P3Oven7].Io.DIONSwitch:=I602[6]	;//	1_3烤箱门打开
arrCyCtrl[P3CYNo.P3Oven10].Io.DIOFFSwitch:=I602[7]	;//	1_4烤箱门关闭
arrCyCtrl[P3CYNo.P3Oven10].Io.DIONSwitch:=I602[8]	;//	1_4烤箱门打开
arrCyCtrl[P3CYNo.P3Oven13].Io.DIOFFSwitch:=I602[9]	;//	1_5烤箱门关闭
arrCyCtrl[P3CYNo.P3Oven13].Io.DIONSwitch:=I602[10] 	;//	1_5烤箱门打开
arrCyCtrl[P3CYNo.P3Oven16].Io.DIOFFSwitch:=I602[11] ;//	1_6烤箱门关闭
arrCyCtrl[P3CYNo.P3Oven16].Io.DIONSwitch:=I602[12] 	;//	1_6烤箱门打开
arrCyCtrl[P3CYNo.P3Oven19].Io.DIOFFSwitch:=I602[13] ;//	1_7烤箱门关闭
arrCyCtrl[P3CYNo.P3Oven19].Io.DIONSwitch:=I602[14] 	;//	1_7烤箱门打开
P3Senser.P3_Ovendoorswitch1:=I602[15]               ;//	烤箱1对射感应
P3Senser.P3_OVenScapegoat1:=I602[16]               ;//烤箱1替罪羊	
		
//I603		
arrCyCtrl[P3CYNo.P3Oven2].Io.DIOFFSwitch:=I603[1]	;//	2_1烤箱门关闭
arrCyCtrl[P3CYNo.P3Oven2].Io.DIONSwitch:=I603[2]	;//	2_1烤箱门打开
arrCyCtrl[P3CYNo.P3Oven5].Io.DIOFFSwitch:=I603[3]	;//	2_2烤箱门关闭
arrCyCtrl[P3CYNo.P3Oven5].Io.DIONSwitch:=I603[4]	;//	2_2烤箱门打开
arrCyCtrl[P3CYNo.P3Oven8].Io.DIOFFSwitch:=I603[5]	;//	2_3烤箱门关闭
arrCyCtrl[P3CYNo.P3Oven8].Io.DIONSwitch:=I603[6]	;//	2_3烤箱门打开
arrCyCtrl[P3CYNo.P3Oven11].Io.DIOFFSwitch:=I603[7]	;//	2_4烤箱门关闭
arrCyCtrl[P3CYNo.P3Oven11].Io.DIONSwitch:=I603[8]	;//	2_4烤箱门打开
arrCyCtrl[P3CYNo.P3Oven14].Io.DIOFFSwitch:=I603[9]	;//	2_5烤箱门关闭
arrCyCtrl[P3CYNo.P3Oven14].Io.DIONSwitch:=I603[10] 	;//	2_5烤箱门打开
arrCyCtrl[P3CYNo.P3Oven17].Io.DIOFFSwitch:=I603[11] ;//	2_6烤箱门关闭
arrCyCtrl[P3CYNo.P3Oven17].Io.DIONSwitch:=I603[12] 	;//	2_6烤箱门打开
arrCyCtrl[P3CYNo.P3Oven20].Io.DIOFFSwitch:=I603[13] ;//	2_7烤箱门关闭
arrCyCtrl[P3CYNo.P3Oven20].Io.DIONSwitch:=I603[14] 	;//	2_7烤箱门打开
P3Senser.P3_Ovendoorswitch2:=I603[15]               ;//	烤箱2对射感应
P3Senser.P3_OVenScapegoat2:=I603[16] 				 ;//烤箱2替罪羊		
		
		
//I604		
arrCyCtrl[P3CYNo.P3Oven3].Io.DIOFFSwitch:=I604[1]	;//	3_1烤箱门关闭
arrCyCtrl[P3CYNo.P3Oven3].Io.DIONSwitch:=I604[2]	;//	3_1烤箱门打开
arrCyCtrl[P3CYNo.P3Oven6].Io.DIOFFSwitch:=I604[3]	;//	3_2烤箱门关闭
arrCyCtrl[P3CYNo.P3Oven6].Io.DIONSwitch:=I604[4]	;//	3_2烤箱门打开
arrCyCtrl[P3CYNo.P3Oven9].Io.DIOFFSwitch:=I604[5]	;//	3_3烤箱门关闭
arrCyCtrl[P3CYNo.P3Oven9].Io.DIONSwitch:=I604[6]	;//	3_3烤箱门打开
arrCyCtrl[P3CYNo.P3Oven12].Io.DIOFFSwitch:=I604[7]	;//	3_4烤箱门关闭
arrCyCtrl[P3CYNo.P3Oven12].Io.DIONSwitch:=I604[8]	;//	3_4烤箱门打开
arrCyCtrl[P3CYNo.P3Oven15].Io.DIOFFSwitch:=I604[9]	;//	3_5烤箱门关闭
arrCyCtrl[P3CYNo.P3Oven15].Io.DIONSwitch:=I604[10] 	;//	3_5烤箱门打开
arrCyCtrl[P3CYNo.P3Oven18].Io.DIOFFSwitch:=I604[11] ;//	3_6烤箱门关闭
arrCyCtrl[P3CYNo.P3Oven18].Io.DIONSwitch:=I604[12] 	;//	3_6烤箱门打开
arrCyCtrl[P3CYNo.P3Oven21].Io.DIOFFSwitch:=I604[13] ;//	3_7烤箱门关闭
arrCyCtrl[P3CYNo.P3Oven21].Io.DIONSwitch:=I604[14] 	;//	3_7烤箱门打开
P3Senser.P3_Ovendoorswitch3:=I604[15]               ;//	烤箱3对射感应
P3Senser.P3_OVenScapegoat3:=I604[16] 				 ;//烤箱3替罪羊		
	


//I605
arrCyCtrl[P3CYNo.P3ShortTest].Io.DIOnSwitch:=I605[1]	    ;//	短路测试夹气缸张开
arrCyCtrl[P3CYNo.P3ShortTest].Io.DIOFFSwitch:=I605[2]	    ;//	短路测试夹气缸缩回
arrCyCtrl[P3CYNo.P3HotPressTensed].Io.DIOnSwitch:=I605[3]	;//	热压麦拉张紧气缸伸出位
arrCyCtrl[P3CYNo.P3HotPressTensed].Io.DIOFFSwitch:=I605[4]	;//	热压麦拉张紧气缸缩回位
P3Senser.P3_HotEmptyPress:=I605[5]	                        ;//	热压防空压感应
P3Senser.P3_HotScapegoat :=I605[6]	                        ;//	热压替罪羊检测
P3Senser.P3_HotMoveOffset_X:=I605[7]	;//	热压上料偏移检测1x
P3Senser.P3_HotMoveOffset_Y:=I605[8]	;//	热压上料偏移检测2x
P3Senser.P3_HotMoveOffset_Z:=I605[9]	;//	热压上料偏移检测3z
arrCyCtrl[P3CYNo.P3CellPushSpin].Io.DIOffSwitch:=I605[10]  ;//	电芯旋转定位气缸伸出位
arrCyCtrl[P3CYNo.P3CellPushSpin].Io.DIOnSwitch:=I605[11]  ;//	电芯旋转定位气缸缩回位	
arrCyCtrl[P3CYNo.P3WeightFeedingClamp].Io.DIOFFSwitch:=I605[12]  ;//称重上料夹张开位
arrCyCtrl[P3CYNo.P3WeightFeedingClamp].Io.DIONSwitch:=I605[13]   ;//称重上料夹闭合位
P3Senser.P3_WeightSensor:=I605[14]      ;//	称重台有料感应
arrCyCtrl[P3CYNo.P3WgightUP].Io.DIOnSwitch:=      I605[15]  ;//	称重上料夹夹电芯气缸张开位
arrCyCtrl[P3CYNo.P3WgightUP].Io.DIOFFSwitch:=I605[16]  ;//	称重上料夹夹电芯气缸闭合位
	

//I606
arrCyCtrl[P3CYNo.P3ThicknessMeasuringSwitch].Io.DIOnSwitch:=I606[1]	;//测厚台切换气缸伸出位
arrCyCtrl[P3CYNo.P3ThicknessMeasuringSwitch].Io.DIOFFSwitch:=I606[2];//	测厚台切换气缸缩回位
arrCyCtrl[P3CYNo.P3ThicknessSupport].Io.DIOnSwitch:=I606[3]	    ;//	测厚台托板气缸伸出
arrCyCtrl[P3CYNo.P3ThicknessSupport].Io.DIOFFSwitch:=I606[4]	;//	测厚台托板气缸缩回
arrCyCtrl[P3CYNo.P3ThicknessPressure].Io.DIOnSwitch:=I606[5]	;//	测厚台压板气缸伸出
arrCyCtrl[P3CYNo.P3ThicknessPressure].Io.DIOFFSwitch:=I606[6]	;//	测厚台压板气缸缩回
P3Senser.P3_ThicknessSensor:=I606[7]	;//	测厚台有料感应
P3Senser.P3_HotOffset_L:=I606[8]	;//	//热压电芯位置检测1
arrCyCtrl[P3CYNo.P3SortClamp].Io.DIOFFSwitch:=I606[9]	  ;//	电芯分选夹张开位
arrCyCtrl[P3CYNo.P3SortClamp].Io.DIOnSwitch:=I606[10]     ;//	电芯分选夹闭合位
arrCyCtrl[P3CYNo.P3SortLifting].Io.DIOFFSwitch:=I606[11]  ;//	电芯分选夹上升位
arrCyCtrl[P3CYNo.P3SortLifting].Io.DIOnSwitch:=I606[12]   ;//	电芯分选夹下降位
arrCyCtrl[P3CYNo.P3SortRotate].Io.DIOFFSwitch:=I606[13]   ;//	电芯分选夹0度位
arrCyCtrl[P3CYNo.P3SortRotate].Io.DIONSwitch:=I606[14]    ;//	电芯分选夹90度位
arrCyCtrl[P3CYNo.P3TapeSpin].Io.DIOnSwitch:=      I606[15]  ;//	流水线下料旋转气缸张开位
arrCyCtrl[P3CYNo.P3TapeSpin].Io.DIOFFSwitch:=I606[16]  ;//	流水线下料旋转气缸闭合位	


//I607	
arrCyCtrl[P3CYNo.P3BoxLock1_NG].Io.DIOnSwitch:=I607[1]	;//	电芯NG1料盒锁定气缸伸出位
arrCyCtrl[P3CYNo.P3BoxLock1_NG].Io.DIOFFSwitch:=I607[2]	;//	电芯NG1料盒锁定气缸缩回位
P3Senser.P3_PoleMotor2_Height:=I607[3]	;//	电芯NG1料盒高度感应
P3Senser.P3_PoleMotor2_Reach:=I607[4]	;//	电芯NG1料盒到位感应
P3Senser.P3_PoleMotor2_P_OT:=I607[5]	;//	电芯NG1料盒顶升电机上限
P3Senser.P3_PoleMotor2_N_OT:=I607[6]	;//	电芯NG1料盒顶升电机下限
arrCyCtrl[P3CYNo.P3BoxLock2_NG].Io.DIOnSwitch:=I607[7]	;//	电芯NG2料盒锁定气缸伸出位
arrCyCtrl[P3CYNo.P3BoxLock2_NG].Io.DIOFFSwitch:=I607[8]	;//	电芯NG2料盒锁定气缸缩回位
P3Senser.P3_PoleMotor3_Height:=I607[9]	;//	电芯NG2料盒高度感应
P3Senser.P3_PoleMotor3_Reach:=I607[10]  ;//	电芯NG2料盒到位感应
P3Senser.P3_PoleMotor3_P_OT:=I607[11]  ;//	电芯NG2料盒顶升电机上限
P3Senser.P3_PoleMotor3_N_OT:=I607[12]  ;//	电芯NG2料盒顶升电机下限
arrCyCtrl[P3CYNo.P3BoxLock3_NG].Io.DIOnSwitch:=I607[13]  ;//	电芯NG3料盒锁定气缸伸出位
arrCyCtrl[P3CYNo.P3BoxLock3_NG].Io.DIOFFSwitch:=I607[14]  ;//	电芯NG3料盒锁定气缸缩回位
P3Senser.P3_PoleMotor4_Height:=I607[15]  ;//	电芯NG3料盒高度感应
P3Senser.P3_PoleMotor4_Reach:=I607[16]  ;//	电芯NG3料盒到位感应


//I608
P3Senser.P3_PoleMotor4_P_OT:=I608[1]	;//	电芯NG3料盒顶升电机上限
P3Senser.P3_PoleMotor4_N_OT:=I608[2]	;//	电芯NG3料盒顶升电机下限
arrCyCtrl[P3CYNo.P3SortPush].Io.DIOFFSwitch:=I608[3]	;//	电芯分选夹夹电芯张开位
arrCyCtrl[P3CYNo.P3SortPush].Io.DIOnSwitch:=I608[4]	;//	电芯分选夹夹电芯夹紧位
arrCyCtrl[P3CYNo.P3BlankingClamp].Io.DIOFFSwitch:=I608[5]	;//	电芯下料夹张开位
arrCyCtrl[P3CYNo.P3BlankingClamp].Io.DIOnSwitch:=I608[6]	;//	电芯下料夹闭合位
arrCyCtrl[P3CYNo.P3BlankingLifting].Io.DIOFFSwitch:=I608[7]	;//	电芯下料夹上升位
arrCyCtrl[P3CYNo.P3BlankingLifting].Io.DIOnSwitch:=I608[8]	;//	电芯下料夹下降位
P3Senser.P3_CacheSensor:=I608[9]	;//贴胶平台有料感应
P3Senser.P3_PoleMotor2_bHave:=I608[10]  ;//电芯NG1料盒有料感应	
P3Senser.P3_PoleMotor3_bHave:=I608[11]  ;//	电芯NG2料盒有料感应
P3Senser.P3_PoleMotor4_bHave:=I608[12]  ;//	电芯NG3料盒有料感应
arrCyCtrl[P3CYNo.P3CellSpin].Io.DIONSwitch:=I608[13]  ;//电芯旋转气缸0°
arrCyCtrl[P3CYNo.P3CellSpin].Io.DIOFFSwitch:=I608[14]  ;//电芯旋转气缸180°
P3Button.LateStop:=I608[15]  ;//急停按钮
arrCyCtrl[P3CYNo.P3TapeVacuo].Io.DIOnSwitch:=I608[16]  ;//	贴胶头真空

//I609
P3Senser.P3_Securitydoorswitch1:=I609[1]	;//外罩门禁1	
P3Senser.P3_Securitydoorswitch2:=I609[2]	;//外罩门禁2
P3Senser.P3_Securitydoorswitch3:=I609[3]	;//外罩门禁3	
P3Senser.P3_Securitydoorswitch4:=I609[4]	;//外罩门禁4	
P3Senser.P3_Securitydoorswitch5:=I609[5]	;//外罩门禁5	
P3Senser.P3_Securitydoorswitch6:=I609[6]	;//外罩门禁6	
P3Senser.P3_Securitydoorswitch7:=I609[7]	;//外罩门禁7
P3Senser.P3_Securitydoorswitch8:=I609[8]	;//外罩门禁8
P3Senser.P3_Securitydoorswitch9:=I609[9]	;//外罩门禁9	
P3Senser.P3_Securitydoorswitch10:=I609[10]  ;//外罩门禁10	
P3Senser.P3_Securitydoorswitch11:=I609[11]  ;//外罩门禁11	
P3Senser.P3_Securitydoorswitch12:=I609[12]  ;//外罩门禁12	
P3Press.Gluebtn:=I609[13]  ;//拉胶按钮
P3Press.Cutbtn:=I609[14]  ;//切胶按钮
P3Press.Readybtn:=I609[15]  ;//	备胶按钮
P3Senser.P3_BuleHavetape:=I609[16]  ;//后段蓝胶胶带有料检测

arrCyCtrl[P3CYNo.P3CellPush].Io.DIOnSwitch:=I701[1]	;//电芯压紧气缸伸出位	
arrCyCtrl[P3CYNo.P3CellPush].Io.DIOFFSwitch:=I701[2]	;//电芯压紧气缸缩回位
arrCyCtrl[P3CYNo.P3CellAdvance].Io.DIOnSwitch:=I701[3]	;//电芯平移气缸伸出位	
arrCyCtrl[P3CYNo.P3CellAdvance].Io.DIOFFSwitch:=I701[4]	;//电芯平移气缸缩回位	
arrCyCtrl[P3CYNo.P3TapePush].Io.DIOnSwitch:=I701[5]	;//贴胶头夹紧气缸伸出位	
arrCyCtrl[P3CYNo.P3TapePush].Io.DIOFFSwitch:=I701[6]	;//贴胶头夹紧气缸缩回位	
arrCyCtrl[P3CYNo.P3TapePull].Io.DIOnSwitch:=I701[7]	;//拉带气缸伸出位
arrCyCtrl[P3CYNo.P3TapePull].Io.DIOFFSwitch:=I701[8]	;//拉带气缸缩回位
arrCyCtrl[P3CYNo.P3TapeLift].Io.DIOnSwitch:=I701[9]	;//拉带升降气缸伸出位	
arrCyCtrl[P3CYNo.P3TapeLift].Io.DIOFFSwitch:=I701[10]  ;//拉带升降气缸缩回位	
arrCyCtrl[P3CYNo.P3TapeCut].Io.DIOnSwitch:=I701[11]  ;//切胶气缸伸出位	
arrCyCtrl[P3CYNo.P3TapeCut].Io.DIOFFSwitch:=I701[12]  ;//切胶气缸缩回位	
arrCyCtrl[P3CYNo.P3GluePush].Io.DIOFFSwitch:=I701[13]  ;//压胶气缸伸出位	
arrCyCtrl[P3CYNo.P3GluePush].Io.DIOnSwitch:=I701[14]  ;//压胶气缸缩回位	
arrCyCtrl[P3CYNo.P3TapeBuffer].Io.DIOnSwitch:=I701[15]  ;//贴胶缓存气缸伸出位	
arrCyCtrl[P3CYNo.P3TapeBuffer].Io.DIOFFSwitch:=I701[16]  ;//贴胶缓存气缸缩回位	


arrCyCtrl[P3CYNo.P3ColdBlow].Io.DIOnSwitch:=arrCyCtrl[P3CYNo.P3ColdBlow].Io.DOStatus1;//冷压吹气
arrCyCtrl[P3CYNo.P3ColdBlow].Io.DIOFFSwitch:=NOT arrCyCtrl[P3CYNo.P3ColdBlow].Io.DOStatus1;//冷压吹气
arrCyCtrl[P3CYNo.P3HotBlow].Io.DIOnSwitch:=arrCyCtrl[P3CYNo.P3ColdBlow].Io.DOStatus1;//热压吹气
arrCyCtrl[P3CYNo.P3HotBlow].Io.DIOFFSwitch:=NOT arrCyCtrl[P3CYNo.P3ColdBlow].Io.DOStatus1;//热压吹气


//新增
arrCyCtrl[P3CYNo.P3_GlueExtend].Io.DIOnSwitch:=I702[1]  ;//二维码蹬胶气缸蹬出
arrCyCtrl[P3CYNo.P3_GlueExtend].Io.DIOFFSwitch:=arrCyCtrl[P3CYNo.P3_GlueExtend].Io.DOStatus2;//二维码蹬胶气缸缩回
arrCyCtrl[P3CYNo.P3_GluePress].Io.DIOnSwitch:=I702[3]  ;//二维码压胶气缸压紧
arrCyCtrl[P3CYNo.P3_GluePress].Io.DIOFFSwitch:=I702[4]  ;//二维码压胶气缸松开
arrCyCtrl[P3CYNo.P3_GlueCut].Io.DIOnSwitch:=I702[5]  ;//二维码切胶气缸切胶
arrCyCtrl[P3CYNo.P3_GlueCut].Io.DIOFFSwitch:=I702[6]  ;//二维码切胶气缸缩回
arrCyCtrl[P3CYNo.P3_GluePull].Io.DIOnSwitch:=I702[7]  ;//二维码拉胶气缸夹紧
arrCyCtrl[P3CYNo.P3_GluePull].Io.DIOFFSwitch:=I702[8]  ;//二维码拉胶气缸松开
arrCyCtrl[P3CYNo.P3_GlueVacuum].Io.DIONSwitch:=I702[9]  ;//	二维码贴胶吸盘真空
P3Senser.P3_IDMark:=I702[10]  ;//二维码胶Mark孔检测
P3Senser.P3_Securitydoorswitch14:=I702[11]  	;//外罩门禁14
P3Senser.P3_IDHavetape:=I702[12]  ;//二维码胶胶卷有料检测
P3Button.IDStickBtn:=I702[13]  ;//二维码备胶按钮
P3Button.IDGluebtn:=I702[14]  ;//二维码拉胶按钮
P3Button.IDCutbtn:=I702[15]  ;//二维码切胶按钮
P3Senser.P3_Securitydoorswitch15:=I702[16]  	;//外罩门禁15
END_ACTION

ACTION P3_LimitSwitch:
//尾段下料

arrAxisCtrl[P3AxisNo.P3M1_ColdpreLine].Io.DigitalInputs;//冷压上料夹平移电机
arrAxisCtrl[P3AxisNo.P3M1_ColdpreLine].Io.biPosLimit:=  arrAxisCtrl[P3AxisNo.P3M1_ColdpreLine].Io.DigitalInputs.16;
arrAxisCtrl[P3AxisNo.P3M1_ColdpreLine].Io.biNegLimit:=  arrAxisCtrl[P3AxisNo.P3M1_ColdpreLine].Io.DigitalInputs.17;
arrAxisCtrl[P3AxisNo.P3M1_ColdpreLine].Io.biHomeSwitch:=arrAxisCtrl[P3AxisNo.P3M1_ColdpreLine].Io.DigitalInputs.17;

arrAxisCtrl[P3AxisNo.P3M1_ColdpreRetracting].Io.DigitalInputs;//冷压上料夹进退电机
arrAxisCtrl[P3AxisNo.P3M1_ColdpreRetracting].Io.biPosLimit:=  arrAxisCtrl[P3AxisNo.P3M1_ColdpreRetracting].Io.DigitalInputs.16;
arrAxisCtrl[P3AxisNo.P3M1_ColdpreRetracting].Io.biNegLimit:=  arrAxisCtrl[P3AxisNo.P3M1_ColdpreRetracting].Io.DigitalInputs.17;
arrAxisCtrl[P3AxisNo.P3M1_ColdpreRetracting].Io.biHomeSwitch:=arrAxisCtrl[P3AxisNo.P3M1_ColdpreRetracting].Io.DigitalInputs.2;

arrAxisCtrl[P3AxisNo.P3M1_ColdpreWhirling].Io.DigitalInputs;//冷压上料夹旋转电机
arrAxisCtrl[P3AxisNo.P3M1_ColdpreWhirling].Io.biPosLimit:=  arrAxisCtrl[P3AxisNo.P3M1_ColdpreWhirling].Io.DigitalInputs.16;
arrAxisCtrl[P3AxisNo.P3M1_ColdpreWhirling].Io.biNegLimit:=  arrAxisCtrl[P3AxisNo.P3M1_ColdpreWhirling].Io.DigitalInputs.2;
arrAxisCtrl[P3AxisNo.P3M1_ColdpreWhirling].Io.biHomeSwitch:=arrAxisCtrl[P3AxisNo.P3M1_ColdpreWhirling].Io.DigitalInputs.2;

arrAxisCtrl[P3AxisNo.P3M1_ColdpreUpDown].Io.DigitalInputs;//冷压上料夹升降电机
arrAxisCtrl[P3AxisNo.P3M1_ColdpreUpDown].Io.biPosLimit:=  arrAxisCtrl[P3AxisNo.P3M1_ColdpreUpDown].Io.DigitalInputs.16;
arrAxisCtrl[P3AxisNo.P3M1_ColdpreUpDown].Io.biNegLimit:=  arrAxisCtrl[P3AxisNo.P3M1_ColdpreUpDown].Io.DigitalInputs.17;
arrAxisCtrl[P3AxisNo.P3M1_ColdpreUpDown].Io.biHomeSwitch:=arrAxisCtrl[P3AxisNo.P3M1_ColdpreUpDown].Io.DigitalInputs.2;

arrAxisCtrl[P3AxisNo.P3M1_ColdpreSupPlateLine].Io.DigitalInputs;//冷压托板开合电机
arrAxisCtrl[P3AxisNo.P3M1_ColdpreSupPlateLine].Io.biPosLimit:=  arrAxisCtrl[P3AxisNo.P3M1_ColdpreSupPlateLine].Io.DigitalInputs.2;
arrAxisCtrl[P3AxisNo.P3M1_ColdpreSupPlateLine].Io.biNegLimit:=  arrAxisCtrl[P3AxisNo.P3M1_ColdpreSupPlateLine].Io.DigitalInputs.7;
arrAxisCtrl[P3AxisNo.P3M1_ColdpreSupPlateLine].Io.biHomeSwitch:=arrAxisCtrl[P3AxisNo.P3M1_ColdpreSupPlateLine].Io.DigitalInputs.7;

arrAxisCtrl[P3AxisNo.P3M1_ColdpreActuated].Io.DigitalInputs;//冷压驱动电机
arrAxisCtrl[P3AxisNo.P3M1_ColdpreActuated].Io.biPosLimit:=  arrAxisCtrl[P3AxisNo.P3M1_ColdpreActuated].Io.DigitalInputs.16;
arrAxisCtrl[P3AxisNo.P3M1_ColdpreActuated].Io.biNegLimit:=  arrAxisCtrl[P3AxisNo.P3M1_ColdpreActuated].Io.DigitalInputs.17;
arrAxisCtrl[P3AxisNo.P3M1_ColdpreActuated].Io.biHomeSwitch:=arrAxisCtrl[P3AxisNo.P3M1_ColdpreActuated].Io.DigitalInputs.17;

arrAxisCtrlV2[P3AxisNo.P3_M2_OvenCarrying].Io.DigitalInputs;//烤箱上料夹搬运电机
arrAxisCtrlV2[P3AxisNo.P3_M2_OvenCarrying].Io.biPosLimit :=  arrAxisCtrlV2[P3AxisNo.P3_M2_OvenCarrying].Io.DigitalInputs.16;
arrAxisCtrlV2[P3AxisNo.P3_M2_OvenCarrying].Io.biNegLimit :=  arrAxisCtrlV2[P3AxisNo.P3_M2_OvenCarrying].Io.DigitalInputs.17;
arrAxisCtrlV2[P3AxisNo.P3_M2_OvenCarrying].Io.biHomeSwitch :=arrAxisCtrlV2[P3AxisNo.P3_M2_OvenCarrying].Io.DigitalInputs.2;

arrAxisCtrlV2[P3AxisNo.P3_M2_OvenRetracting].Io.DigitalInputs;//烤箱上料夹进退电机
arrAxisCtrlV2[P3AxisNo.P3_M2_OvenRetracting].Io.biPosLimit := arrAxisCtrlV2[P3AxisNo.P3_M2_OvenRetracting].Io.DigitalInputs.16;
//arrAxisCtrlV2[P3AxisNo.P3_M2_OvenRetracting].Io.biNegLimit :=  arrAxisCtrlV2[P3AxisNo.P3_M2_OvenRetracting].Io.DigitalInputs.17;
arrAxisCtrlV2[P3AxisNo.P3_M2_OvenRetracting].Io.biHomeSwitch := arrAxisCtrlV2[P3AxisNo.P3_M2_OvenRetracting].Io.DigitalInputs.17;

arrAxisCtrlV2[P3AxisNo.P3_M2_OvenUpDown].Io.DigitalInputs;//烤箱上料夹升降电机
arrAxisCtrlV2[P3AxisNo.P3_M2_OvenUpDown].Io.biPosLimit:=  arrAxisCtrlV2[P3AxisNo.P3_M2_OvenUpDown].Io.DigitalInputs.16;
arrAxisCtrlV2[P3AxisNo.P3_M2_OvenUpDown].Io.biNegLimit:=  arrAxisCtrlV2[P3AxisNo.P3_M2_OvenUpDown].Io.DigitalInputs.17;
arrAxisCtrlV2[P3AxisNo.P3_M2_OvenUpDown].Io.biHomeSwitch:= arrAxisCtrlV2[P3AxisNo.P3_M2_OvenUpDown].Io.DigitalInputs.2;

arrAxisCtrl[P3AxisNo.P3_M3_HotPressingActuated].Io.DigitalInputs;//热压驱动电机
arrAxisCtrl[P3AxisNo.P3_M3_HotPressingActuated].Io.biPosLimit:=  arrAxisCtrl[P3AxisNo.P3_M3_HotPressingActuated].Io.DigitalInputs.16;
arrAxisCtrl[P3AxisNo.P3_M3_HotPressingActuated].Io.biNegLimit:=  arrAxisCtrl[P3AxisNo.P3_M3_HotPressingActuated].Io.DigitalInputs.17;
arrAxisCtrl[P3AxisNo.P3_M3_HotPressingActuated].Io.biHomeSwitch:=arrAxisCtrl[P3AxisNo.P3_M3_HotPressingActuated].Io.DigitalInputs.17;

arrAxisCtrl[P3AxisNo.P3_M3_HotPressingLine].Io.DigitalInputs;//热压托板开合电机
arrAxisCtrl[P3AxisNo.P3_M3_HotPressingLine].Io.biPosLimit:=  arrAxisCtrl[P3AxisNo.P3_M3_HotPressingLine].Io.DigitalInputs.2;
arrAxisCtrl[P3AxisNo.P3_M3_HotPressingLine].Io.biNegLimit:=  arrAxisCtrl[P3AxisNo.P3_M3_HotPressingLine].Io.DigitalInputs.7;
arrAxisCtrl[P3AxisNo.P3_M3_HotPressingLine].Io.biHomeSwitch:=arrAxisCtrl[P3AxisNo.P3_M3_HotPressingLine].Io.DigitalInputs.7;

arrAxisCtrl[P3AxisNo.P3_M4_OffloadingCarrying].Io.DigitalInputs;//电芯下料夹搬运电机
arrAxisCtrl[P3AxisNo.P3_M4_OffloadingCarrying].Io.biPosLimit:=  arrAxisCtrl[P3AxisNo.P3_M4_OffloadingCarrying].Io.DigitalInputs.16;
arrAxisCtrl[P3AxisNo.P3_M4_OffloadingCarrying].Io.biNegLimit:=  arrAxisCtrl[P3AxisNo.P3_M4_OffloadingCarrying].Io.DigitalInputs.17;
arrAxisCtrl[P3AxisNo.P3_M4_OffloadingCarrying].Io.biHomeSwitch:=arrAxisCtrl[P3AxisNo.P3_M4_OffloadingCarrying].Io.DigitalInputs.17;

arrAxisCtrl[P3AxisNo.P3_M4_OffloadingUpDown].Io.DigitalInputs;//电芯下料夹升降电机
arrAxisCtrl[P3AxisNo.P3_M4_OffloadingUpDown].Io.biPosLimit:=  arrAxisCtrl[P3AxisNo.P3_M4_OffloadingUpDown].Io.DigitalInputs.16;
arrAxisCtrl[P3AxisNo.P3_M4_OffloadingUpDown].Io.biNegLimit:=  arrAxisCtrl[P3AxisNo.P3_M4_OffloadingUpDown].Io.DigitalInputs.17;
arrAxisCtrl[P3AxisNo.P3_M4_OffloadingUpDown].Io.biHomeSwitch:=arrAxisCtrl[P3AxisNo.P3_M4_OffloadingUpDown].Io.DigitalInputs.2;

arrAxisCtrl[P3AxisNo.P3_M4_SortingoutCarrying].Io.DigitalInputs;//电芯分选夹搬运电机
arrAxisCtrl[P3AxisNo.P3_M4_SortingoutCarrying].Io.biPosLimit:=  arrAxisCtrl[P3AxisNo.P3_M4_SortingoutCarrying].Io.DigitalInputs.16;
arrAxisCtrl[P3AxisNo.P3_M4_SortingoutCarrying].Io.biNegLimit:=  arrAxisCtrl[P3AxisNo.P3_M4_SortingoutCarrying].Io.DigitalInputs.17;
arrAxisCtrl[P3AxisNo.P3_M4_SortingoutCarrying].Io.biHomeSwitch:=arrAxisCtrl[P3AxisNo.P3_M4_SortingoutCarrying].Io.DigitalInputs.17;

arrAxisCtrl[P3AxisNo.P3_M4_SortingoutUpDown].Io.DigitalInputs;//电芯分选夹升降电机
arrAxisCtrl[P3AxisNo.P3_M4_SortingoutUpDown].Io.biPosLimit:=  arrAxisCtrl[P3AxisNo.P3_M4_SortingoutUpDown].Io.DigitalInputs.16;
arrAxisCtrl[P3AxisNo.P3_M4_SortingoutUpDown].Io.biNegLimit:=  arrAxisCtrl[P3AxisNo.P3_M4_SortingoutUpDown].Io.DigitalInputs.17;
arrAxisCtrl[P3AxisNo.P3_M4_SortingoutUpDown].Io.biHomeSwitch:=arrAxisCtrl[P3AxisNo.P3_M4_SortingoutUpDown].Io.DigitalInputs.2;

arrAxisCtrl[P3AxisNo.P3_M4_WeighLine].Io.DigitalInputs;//称重上料夹平移电机
arrAxisCtrl[P3AxisNo.P3_M4_WeighLine].Io.biPosLimit:=  arrAxisCtrl[P3AxisNo.P3_M4_WeighLine].Io.DigitalInputs.16;
arrAxisCtrl[P3AxisNo.P3_M4_WeighLine].Io.biNegLimit:=  arrAxisCtrl[P3AxisNo.P3_M4_WeighLine].Io.DigitalInputs.17;
arrAxisCtrl[P3AxisNo.P3_M4_WeighLine].Io.biHomeSwitch:=arrAxisCtrl[P3AxisNo.P3_M4_WeighLine].Io.DigitalInputs.17;

arrAxisCtrl[P3AxisNo.P3_M4_WeighUpDown].Io.DigitalInputs;//称重上料夹升降电机
arrAxisCtrl[P3AxisNo.P3_M4_WeighUpDown].Io.biPosLimit:=  arrAxisCtrl[P3AxisNo.P3_M4_WeighUpDown].Io.DigitalInputs.16;
arrAxisCtrl[P3AxisNo.P3_M4_WeighUpDown].Io.biNegLimit:=  arrAxisCtrl[P3AxisNo.P3_M4_WeighUpDown].Io.DigitalInputs.17;
arrAxisCtrl[P3AxisNo.P3_M4_WeighUpDown].Io.biHomeSwitch:=arrAxisCtrl[P3AxisNo.P3_M4_WeighUpDown].Io.DigitalInputs.2;

arrAxisCtrl[P3AxisNo.P3_M4_WeighWhirling].Io.DigitalInputs;//称重上料夹旋转电机
arrAxisCtrl[P3AxisNo.P3_M4_WeighWhirling].Io.biPosLimit:=  FALSE;
arrAxisCtrl[P3AxisNo.P3_M4_WeighWhirling].Io.biNegLimit:=  FALSE;
arrAxisCtrl[P3AxisNo.P3_M4_WeighWhirling].Io.biHomeSwitch:=arrAxisCtrl[P3AxisNo.P3_M4_WeighWhirling].Io.DigitalInputs.2;

arrAxisCtrl[P3AxisNo.P3_TapeAdvance].Io.DigitalInputs;//贴胶头进退
arrAxisCtrl[P3AxisNo.P3_TapeAdvance].Io.biPosLimit:=  arrAxisCtrl[P3AxisNo.P3_TapeAdvance].Io.DigitalInputs.16;
arrAxisCtrl[P3AxisNo.P3_TapeAdvance].Io.biNegLimit:=  arrAxisCtrl[P3AxisNo.P3_TapeAdvance].Io.DigitalInputs.17;
arrAxisCtrl[P3AxisNo.P3_TapeAdvance].Io.biHomeSwitch:=arrAxisCtrl[P3AxisNo.P3_TapeAdvance].Io.DigitalInputs.2;

arrAxisCtrl[P3AxisNo.P3_TapeTranslation].Io.DigitalInputs;//贴胶平移
arrAxisCtrl[P3AxisNo.P3_TapeTranslation].Io.biPosLimit:=  arrAxisCtrl[P3AxisNo.P3_TapeTranslation].Io.DigitalInputs.16;
arrAxisCtrl[P3AxisNo.P3_TapeTranslation].Io.biNegLimit:=  arrAxisCtrl[P3AxisNo.P3_TapeTranslation].Io.DigitalInputs.17;
arrAxisCtrl[P3AxisNo.P3_TapeTranslation].Io.biHomeSwitch:=arrAxisCtrl[P3AxisNo.P3_TapeTranslation].Io.DigitalInputs.2;

arrAxisCtrl[P3AxisNo.P3_IDPut].Io.DigitalInputs;//二维码胶拉胶
arrAxisCtrl[P3AxisNo.P3_IDPut].Io.biPosLimit:=  arrAxisCtrl[P3AxisNo.P3_IDPut].Io.DigitalInputs.16;
arrAxisCtrl[P3AxisNo.P3_IDPut].Io.biNegLimit:=  arrAxisCtrl[P3AxisNo.P3_IDPut].Io.DigitalInputs.17;
arrAxisCtrl[P3AxisNo.P3_IDPut].Io.biHomeSwitch:=arrAxisCtrl[P3AxisNo.P3_IDPut].Io.DigitalInputs.2;

arrAxisCtrl[P3AxisNo.P3_IDLift].Io.DigitalInputs;//二维码胶升降
arrAxisCtrl[P3AxisNo.P3_IDLift].Io.biPosLimit:=  arrAxisCtrl[P3AxisNo.P3_IDLift].Io.DigitalInputs.16;
arrAxisCtrl[P3AxisNo.P3_IDLift].Io.biNegLimit:=  arrAxisCtrl[P3AxisNo.P3_IDLift].Io.DigitalInputs.17;
arrAxisCtrl[P3AxisNo.P3_IDLift].Io.biHomeSwitch:=arrAxisCtrl[P3AxisNo.P3_IDLift].Io.DigitalInputs.2;
END_ACTION

ACTION P3_OutPut:
//尾段下料
Q601[1]:=arrCyCtrl[P3CYNo.P3ColdPressTensed].Io.DOStatus2	;//	冷压麦拉张紧气缸伸出
Q601[2]:=arrCyCtrl[P3CYNo.P3ColdPressTensed].Io.DOStatus1	;//	冷压麦拉张紧气缸缩回
Q601[3]	:=P3Senser.P3_Cold_clear;//	冷压清零
Q601[4]	:=P3Senser.P3_Hot_clear;//	   热压清零
Q601[5]:=arrCyCtrl[P3CYNo.P3OvenMoveClip].Io.DOStatus2	;//	烤箱上料夹张开
Q601[6]:=arrCyCtrl[P3CYNo.P3OvenMoveClip].Io.DOStatus1	;//	烤箱上料夹闭合
Q601[7]:=P3Senser.P3_ShortTest_Start 	;//	短路测试测量开始

Q601[8]:=arrCyCtrl[P3CYNo.P3ColdBlow].Io.DOStatus1	;//冷压吹气
Q601[9]:=arrCyCtrl[P3CYNo.P3HotBlow].Io.DOStatus1	;//热压吹气

Q601[10]:=P3Senser.P3_Tricolorlamp_Yellow;//	后段三色灯-黄
Q601[11]:=P3Senser.P3_Tricolorlamp_Green;//	后段三色灯-绿
Q601[12]:=P3Senser.P3_Tricolorlamp_Red;//	后段三色灯-红
Q601[13]:=P3Senser.P3_Tricolorlamp_Buzzer;//	后段三色灯-蜂鸣器
Q601[14];//	
Q601[15]:=P3Senser.P3_OutSafe;//下料位置安全	
Q601[16]:=P3Senser.P3_OutSendFinish;//	下料放料完成



Q602[1]:=arrCyCtrl[P3CYNo.P3Oven1].Io.DOStatus1	  ;//	1_1烤箱托板上升
Q602[2]:=arrCyCtrl[P3CYNo.P3Oven1].Io.DOStatus2	  ;//	1_1烤箱托板下降
Q602[3]:=arrCyCtrl[P3CYNo.P3Oven4].Io.DOStatus1	  ;//	1_2烤箱托板上升
Q602[4]:=arrCyCtrl[P3CYNo.P3Oven4].Io.DOStatus2	  ;//	1_2烤箱托板下降
Q602[5]:=arrCyCtrl[P3CYNo.P3Oven7].Io.DOStatus1	  ;//	1_3烤箱托板上升
Q602[6]:=arrCyCtrl[P3CYNo.P3Oven7].Io.DOStatus2	  ;//	1_3烤箱托板下降
Q602[7]:=arrCyCtrl[P3CYNo.P3Oven10].Io.DOStatus1  ;//	1_4烤箱托板上升
Q602[8]:=arrCyCtrl[P3CYNo.P3Oven10].Io.DOStatus2  ;//	1_4烤箱托板下降
Q602[9]:=arrCyCtrl[P3CYNo.P3Oven13].Io.DOStatus1  ;//	1_5烤箱托板上升
Q602[10]:=arrCyCtrl[P3CYNo.P3Oven13].Io.DOStatus2 ;//	1_5烤箱托板下降
Q602[11]:=arrCyCtrl[P3CYNo.P3Oven16].Io.DOStatus1 ;//	1_6烤箱托板上升
Q602[12]:=arrCyCtrl[P3CYNo.P3Oven16].Io.DOStatus2 ;//	1_6烤箱托板下降
Q602[13]:=arrCyCtrl[P3CYNo.P3Oven19].Io.DOStatus1 ;//	1_7烤箱托板上升
Q602[14]:=arrCyCtrl[P3CYNo.P3Oven19].Io.DOStatus2 ;//	1_7烤箱托板下降
Q602[15];//	
Q602[16];//	
	
Q603[1]:=arrCyCtrl[P3CYNo.P3Oven2].Io.DOStatus1	  ;//	2_1烤箱托板上升
Q603[2]:=arrCyCtrl[P3CYNo.P3Oven2].Io.DOStatus2   ;//	2_1烤箱托板下降
Q603[3]:=arrCyCtrl[P3CYNo.P3Oven5].Io.DOStatus1	  ;//	2_2烤箱托板上升
Q603[4]:=arrCyCtrl[P3CYNo.P3Oven5].Io.DOStatus2	  ;//	2_2烤箱托板下降
Q603[5]:=arrCyCtrl[P3CYNo.P3Oven8].Io.DOStatus1   ;//	2_3烤箱托板上升
Q603[6]:=arrCyCtrl[P3CYNo.P3Oven8].Io.DOStatus2	  ;//	2_3烤箱托板下降
Q603[7]:=arrCyCtrl[P3CYNo.P3Oven11].Io.DOStatus1  ;//	2_4烤箱托板上升
Q603[8]:=arrCyCtrl[P3CYNo.P3Oven11].Io.DOStatus2  ;//	2_4烤箱托板下降
Q603[9]:=arrCyCtrl[P3CYNo.P3Oven14].Io.DOStatus1  ;//	2_5烤箱托板上升
Q603[10]:=arrCyCtrl[P3CYNo.P3Oven14].Io.DOStatus2 ;//	2_5烤箱托板下降
Q603[11]:=arrCyCtrl[P3CYNo.P3Oven17].Io.DOStatus1 ;//	2_6烤箱托板上升
Q603[12]:=arrCyCtrl[P3CYNo.P3Oven17].Io.DOStatus2 ;//	2_6烤箱托板下降
Q603[13]:=arrCyCtrl[P3CYNo.P3Oven20].Io.DOStatus1 ;//	2_7烤箱托板上升
Q603[14]:=arrCyCtrl[P3CYNo.P3Oven20].Io.DOStatus2 ;//	2_7烤箱托板下降
Q603[15];//	
Q603[16];//	

Q604[1]:=arrCyCtrl[P3CYNo.P3Oven3].Io.DOStatus1	  ;//	3_1烤箱托板上升
Q604[2]:=arrCyCtrl[P3CYNo.P3Oven3].Io.DOStatus2	  ;//	3_1烤箱托板下降
Q604[3]:=arrCyCtrl[P3CYNo.P3Oven6].Io.DOStatus1   ;//	3_2烤箱托板上升
Q604[4]:=arrCyCtrl[P3CYNo.P3Oven6].Io.DOStatus2	  ;//	3_2烤箱托板下降
Q604[5]:=arrCyCtrl[P3CYNo.P3Oven9].Io.DOStatus1	  ;//	3_3烤箱托板上升
Q604[6]:=arrCyCtrl[P3CYNo.P3Oven9].Io.DOStatus2	  ;//	3_3烤箱托板下降
Q604[7]:=arrCyCtrl[P3CYNo.P3Oven12].Io.DOStatus1  ;//	3_4烤箱托板上升
Q604[8]:=arrCyCtrl[P3CYNo.P3Oven12].Io.DOStatus2  ;//	3_4烤箱托板下降
Q604[9]:=arrCyCtrl[P3CYNo.P3Oven15].Io.DOStatus1  ;//	3_5烤箱托板上升
Q604[10]:=arrCyCtrl[P3CYNo.P3Oven15].Io.DOStatus2 ;//	3_5烤箱托板下降
Q604[11]:=arrCyCtrl[P3CYNo.P3Oven18].Io.DOStatus1 ;//	3_6烤箱托板上升
Q604[12]:=arrCyCtrl[P3CYNo.P3Oven18].Io.DOStatus2 ;//	3_6烤箱托板下降
Q604[13]:=arrCyCtrl[P3CYNo.P3Oven21].Io.DOStatus1 ;//	3_7烤箱托板上升
Q604[14]:=arrCyCtrl[P3CYNo.P3Oven21].Io.DOStatus2 ;//	3_7烤箱托板下降
Q604[15];//	
Q604[16];//	

Q605[1]:=arrCyCtrl[P3CYNo.P3ShortTest].Io.DOStatus2	;//	短路测试夹气缸张开
Q605[2]:=arrCyCtrl[P3CYNo.P3ShortTest].Io.DOStatus1	;//	短路测试夹气缸缩回
Q605[3]:=arrCyCtrl[P3CYNo.P3HotPressTensed].Io.DOStatus2	;//	热压麦拉张紧气缸伸出
Q605[4]:=arrCyCtrl[P3CYNo.P3HotPressTensed].Io.DOStatus1	;//	热压麦拉张紧气缸缩回
Q605[5]	;//	
Q605[6]	;//	
Q605[7]	;//	
Q605[8] :=P3Senser.P3_Oven_Power1		;//	
Q605[9]	:=P3Senser.P3_Hotpress_Power		;//	
Q605[10];//	
Q605[11];//	
Q605[12]:=arrCyCtrl[P3CYNo.P3WeightFeedingClamp].Io.DOStatus1;//	称重上料夹张开
Q605[13]:=arrCyCtrl[P3CYNo.P3WeightFeedingClamp].Io.DOStatus2;//	称重上料夹闭合
Q605[14];//	
Q605[15]:=arrCyCtrl[P3CYNo.P3WgightUP].Io.DOStatus1;//	
Q605[16]:=arrCyCtrl[P3CYNo.P3SortPush].Io.DOStatus1;//	

Q606[1]:=arrCyCtrl[P3CYNo.P3ThicknessMeasuringSwitch].Io.DOStatus2	;//	测厚台切换气缸伸出
Q606[2]:=arrCyCtrl[P3CYNo.P3ThicknessMeasuringSwitch].Io.DOStatus1	;//	测厚台切换气缸缩回
Q606[3]:=arrCyCtrl[P3CYNo.P3ThicknessSupport].Io.DOStatus2	;//	测厚台托板气缸伸出
Q606[4]:=arrCyCtrl[P3CYNo.P3ThicknessSupport].Io.DOStatus1	;//	测厚台托板气缸缩回
Q606[5]:=arrCyCtrl[P3CYNo.P3ThicknessPressure].Io.DOStatus2	;//	测厚台压板气缸伸出
Q606[6]:=arrCyCtrl[P3CYNo.P3ThicknessPressure].Io.DOStatus1	;//	测厚台压板气缸缩回
Q606[7]	;//	
Q606[8]	;//	
Q606[9]:=arrCyCtrl[P3CYNo.P3SortClamp].Io.DOStatus1	;//	电芯分选夹张开
Q606[10]:=arrCyCtrl[P3CYNo.P3SortClamp].Io.DOStatus2;//	电芯分选夹闭合
Q606[11]:=arrCyCtrl[P3CYNo.P3SortLifting].Io.DOStatus1;//	电芯分选夹上升
Q606[12]:=arrCyCtrl[P3CYNo.P3SortLifting].Io.DOStatus2;//	电芯分选夹下降
Q606[13]:=arrCyCtrl[P3CYNo.P3SortRotate].Io.DOStatus1;//	电芯分选夹旋转0度
Q606[14]:=arrCyCtrl[P3CYNo.P3SortRotate].Io.DOStatus2;//	电芯分选夹旋转90度
Q606[15]:=arrCyCtrl[P3CYNo.P3TapeSpin].Io.DOStatus1	;//贴胶旋转气缸伸出位;//	
Q606[16]:=arrCyCtrl[P3CYNo.P3TapeSpin].Io.DOStatus2	;//贴胶旋转气缸缩回位	;//	

Q607[1]:=arrCyCtrl[P3CYNo.P3BoxLock1_NG].Io.DOStatus2	;//	电芯NG1料盒锁定气缸伸出
Q607[2]:=arrCyCtrl[P3CYNo.P3BoxLock1_NG].Io.DOStatus1	;//	电芯NG1料盒锁定气缸缩回
Q607[3]:=P3Senser.P3_PoleMotor2_JogP	;//	NG料盒1排杆电机正转
Q607[4]:=P3Senser.P3_PoleMotor2_JogN 	;//	NG料盒1排杆电机反转
Q607[5]:=arrCyCtrl[P3CYNo.P3BoxLock2_NG].Io.DOStatus2	;//	电芯NG2料盒锁定气缸伸出
Q607[6]:=arrCyCtrl[P3CYNo.P3BoxLock2_NG].Io.DOStatus1	;//	电芯NG2料盒锁定气缸缩回
Q607[7]:=P3Senser.P3_PoleMotor3_JogP	;//	NG料盒2排杆电机正转
Q607[8]:=P3Senser.P3_PoleMotor3_JogN	;//	NG料盒2排杆电机反转
Q607[9]:=arrCyCtrl[P3CYNo.P3BoxLock3_NG].Io.DOStatus2	;//	电芯NG3料盒锁定气缸伸出
Q607[10]:=arrCyCtrl[P3CYNo.P3BoxLock3_NG].Io.DOStatus1  ;//	电芯NG3料盒锁定气缸缩回
Q607[11]:=P3Senser.P3_PoleMotor4_JogP   ;//	NG料盒3排杆电机正转
Q607[12]:=P3Senser.P3_PoleMotor4_JogN;//	NG料盒3排杆电机反转
Q607[13];//	
Q607[14];//	
Q607[15];//	
Q607[16];//	



Q608[1]:=arrCyCtrl[P3CYNo.P3CellPushSpin].Io.DOStatus1		;//P3电芯旋转定位气缸 
Q608[2]:=arrCyCtrl[P3CYNo.P3CellPush].Io.DOStatus1			;//P3电芯压紧气缸
Q608[3]:=arrCyCtrl[P3CYNo.P3BlankingRotate].Io.DOStatus1	;//	电芯下料夹旋转0度
Q608[4]:=arrCyCtrl[P3CYNo.P3BlankingRotate].Io.DOStatus2	;//	电芯下料夹旋转90度
Q608[5]:=arrCyCtrl[P3CYNo.P3BlankingClamp].Io.DOStatus1	    ;//	电芯下料夹张开
Q608[6]:=arrCyCtrl[P3CYNo.P3BlankingClamp].Io.DOStatus2		;//	电芯下料夹闭合
Q608[7]:=arrCyCtrl[P3CYNo.P3BlankingLifting].Io.DOStatus1		;//	电芯下料夹上升
Q608[8]:=arrCyCtrl[P3CYNo.P3BlankingLifting].Io.DOStatus2		;//	电芯下料夹下降
Q608[9]	:=arrCyCtrl[P3CYNo.P3_GlueExtend].Io.DOStatus1;//二维码蹬胶气缸
Q608[10]:=arrCyCtrl[P3CYNo.P3_GluePress].Io.DOStatus1;//二维码压胶气缸
Q608[11]:=arrCyCtrl[P3CYNo.P3_GlueCut].Io.DOStatus1;//	二维码切胶气缸
Q608[12]:=arrCyCtrl[P3CYNo.P3_GluePull].Io.DOStatus1;//二维码拉胶气缸夹紧	
Q608[13]:=arrCyCtrl[P3CYNo.P3TapeSpin].Io.DOStatus1	;//贴胶旋转气缸伸出位	
Q608[14]:=arrCyCtrl[P3CYNo.P3TapeSpin].Io.DOStatus2;//	贴胶旋转气缸缩回位
Q608[15]:=arrCyCtrl[P3CYNo.P3TapeVacuo].Io.DOStatus1;//贴胶头真空开
Q608[16]:=arrCyCtrl[P3CYNo.P3_GlueVacuum].Io.DOStatus1;//		二维码贴胶吸盘真空



Q609[1]:=arrCyCtrl[P3CYNo.P3CellSpin].Io.DOStatus1	;//P3电芯旋转气缸伸出位	
Q609[2]:=arrCyCtrl[P3CYNo.P3CellSpin].Io.DOStatus2	;//P3电芯旋转气缸缩回位	
Q609[3]:=arrCyCtrl[P3CYNo.P3CellAdvance].Io.DOStatus1	;//电芯平移气缸伸出位	
Q609[4]	:=arrCyCtrl[P3CYNo.P3CellAdvance].Io.DOStatus2;//	电芯平移气缸缩回位
Q609[5]:=arrCyCtrl[P3CYNo.P3TapePush].Io.DOStatus1	;//贴胶头夹紧气缸伸出位
Q609[6]:=arrCyCtrl[P3CYNo.P3TapePush].Io.DOStatus2	;//贴胶头夹紧气缸缩回位
Q609[7]:=arrCyCtrl[P3CYNo.P3TapePull].Io.DOStatus1	;//拉带夹紧气缸伸出位	
Q609[8]:=arrCyCtrl[P3CYNo.P3TapePull].Io.DOStatus2	;//拉带夹紧气缸缩回位	
Q609[9]:=arrCyCtrl[P3CYNo.P3TapeLift].Io.DOStatus1	;//拉带升降气缸伸出位	
Q609[10]:=arrCyCtrl[P3CYNo.P3TapeLift].Io.DOStatus2;//	拉带升降气缸缩回位
Q609[11]:=arrCyCtrl[P3CYNo.P3TapeCut].Io.DOStatus1;//	切胶气缸伸出位
Q609[12]:=arrCyCtrl[P3CYNo.P3TapeCut].Io.DOStatus2;//	切胶气缸缩回位
Q609[13]:=arrCyCtrl[P3CYNo.P3GluePush].Io.DOStatus1;//压胶气缸伸出位	
Q609[14]:=arrCyCtrl[P3CYNo.P3GluePush].Io.DOStatus2;//	压胶气缸缩回位
Q609[15]:=arrCyCtrl[P3CYNo.P3TapeBuffer].Io.DOStatus1;//	贴胶缓存气缸伸出位
Q609[16]:=arrCyCtrl[P3CYNo.P3TapeBuffer].Io.DOStatus2;//	贴胶缓存气缸缩回位
END_ACTION

END_PROGRAM

// ---- P3POUs/POUs/P3MainState.TcPOU
PROGRAM P3MainState
VAR
	iMainSetp :INT;
	bEstop: BOOL;

	I1: UINT;
	iErrorSetp: INT;
	iLightSel: INT;
	bTurnOn: BOOL;
	bDoor_Stop: BOOL;
	I2: INT;
	I4: INT;
	I5: INT;
	i: UINT;
	iCode2: ICode;
	ExtSetVel: LREAL;
	ExtSetPos: LREAL;
	ExtSetAcc: LREAL;
	ExtSetDec: DINT;
	InitSetp: INT;
	rtStoping: R_TRIG;
	iMainInitSetp: INT;
	iMainEStopSetp: INT;
	K1: UINT;
	bInitReset: BOOL;
	DA1: INT;
	Code1: BOOL;
	Code2: BOOL;
	Code3: BOOL;
	Code4: BOOL;
	CyCtrl: INT;
	bWaterOn: BOOL;
	
	Execute: BOOL;
	bCoeWrite_GlueFeed: BOOL;
	bWaterOn2: BOOL;
	
	P2M1_tonEStop1: INT;
	IN: INT;
	tCycleTimer: TON;
	bSave: BOOL;
	rt10: R_TRIG;
	bReadDataFirstCyle: BOOL;
	testii: INT;
	bSaveDataTest: BOOL;
	testii2: INT;
	bReadDataCyle2: BOOL;
	rtSaveData: R_TRIG;
END_VAR

VAR
	iMainSetp_TON :ARRAY[1..5] OF TON;
	R_TRIG_Bt: 			ARRAY[1..10]OF R_TRIG;
	TON20:Tc2_Standard.TON;	
//	TON21:Tc2_Standard.TON;	
	rt100:Tc2_Standard.R_TRIG;
	rt101:Tc2_Standard.R_TRIG;
	
	tDelayBuzze:TON;

	RT200:ARRAY[1..4] OF Tc2_Standard.R_TRIG;

	csAxis                 :ARRAY[160..185] OF   CS_AxisCtrl;
	csAxisV2               :ARRAY[166..168] OF     CS_AxisCtrlV2;
	fbCy                   :ARRAY[230..289]    OF   FB_Cylinder;
  //  fbRec                 :ARRAY[1..MaxRec]   OF   FB_Rectify;
    fbTemp             :ARRAY[1..MaxTemp]   OF   FB_Temperature;



    csCodeTcp:CS_CodeTcp;
    fbCamInTest: MC_CamIn;//主轴与驱动凸轮耦合

//速度模式验证
	MC_ExtSetPointGenDisable: MC_ExtSetPointGenDisable;
	MC_ExtSetPointGenEnable: MC_ExtSetPointGenEnable;
    MC_ExtSetPointGenOut:        Tc2_MC2.ST_McOutputs;
    MC_ExtSetPointGenOut2:        Tc2_MC2.ST_McOutputs;

    tonEStop:                     Tc2_Standard.TON;

   
  fbP4NGSetpMoter  : CS_SetpMoter;
 


mc_Home    :MC_Home;

     fbCoeWrite_GlueFeed:       FB_EcCoeSdoWrite;
     	wEncodeHome                    :WORD:=6;
        //fbDataXML  :FB_DataXMLP3;  
	rMES:ARRAY[1..20]OF R_TRIG;//
	tMES:ARRAY[1..10]OF TON;//
END_VAR

P3_SystemRUN.btnAuto;
P3_SystemRUN.btnManul;
P3_SystemRUN.btnStart;
P3_SystemRUN.btnStop;
P3_SystemRUN.btnReset;
P3_SystemRUN.btnEstop;//常开  




IF P3_SystemRUN.hmiAuto AND P3Button.P3_Autobtn THEN
	P3_SystemRUN.FlgManua:=FALSE;//尾端下料手动标志
	P3_SystemRUN.FlgAuto:=TRUE;//尾端下料自动标志
ELSE
	P3_SystemRUN.FlgManua:=TRUE;//尾端下料手动标志
	P3_SystemRUN.FlgAuto:=FALSE;///尾端下料自动标志
END_IF


R_TRIG_Bt[1](CLK:=  P3_SystemRUN.hmiStart (*OR P3Button.P3_Startbtn*) );
R_TRIG_Bt[7](CLK:=P3_SystemRUN.btnReset OR  P3_SystemRUN.hmiReset OR stSysState.hmiReset OR P3Button.P3_Resetebtn);
P3_SystemRUN.bReset:=R_TRIG_Bt[7].Q  OR  bInitReset    ;  //复位



//尾段急停
IF   P3_SystemRUN.btnStop OR NOT P3Button.LateStop THEN
	iMainSetp:=400;     
END_IF

IF R_TRIG_Bt[7].Q THEN
	FOR i:=160 TO 177 DO
		HMI_TorAlarm_D[i]:=FALSE;//扭矩报警复位
	END_FOR
END_IF



CASE  iMainSetp OF
		0://   INIT
			Init();
			P3_SystemRUN.iMode:=0;
		 IF  P3_SystemRUN.bInitDone THEN
			 iMainSetp:=88;	
		  END_IF
		88://切换手动
		  IF  P3_SystemRUN.FlgManua OR P3_SystemRUN.btnStop THEN
			  iMainSetp:=300;
		  END_IF
		 
		300://手动状态
				P3_SystemRUN.iMode:=3;//手动状态
				iMainSetp:=310;
		310://等待切换到自动启动  
				IF  P3_SystemRUN.hmiAuto AND NOT P3_SystemRUN.btnStop AND NOT b_Alarm[4]THEN//在自动下、在轴回原点完成、没有报警
							IF R_TRIG_Bt[1].Q THEN
								P3_SystemRUN.iMode:=1;//自动状态
								iMainSetp:=320;
							END_IF
				END_IF
		320://判断是否切换到手动、是否有报警，则切换到手动
				IF NOT P3_SystemRUN.hmiAuto OR P3_SystemRUN.hmiStop  OR  b_Alarm[4] OR P3Button.P3_Stopbtn THEN//
					P3_SystemRUN.hmiAuto:=FALSE;
					iMainSetp:=300;
				END_IF
 (************************急停********************************) 
		400://Stoping
		   P3_SystemRUN.iMode:=4;
			EStop();  
		   iMainSetp:=450;  
			  
		450: //急停跳出 
			IF  NOT  P3_SystemRUN.btnEstop   THEN  
				iMainSetp_TON[2](IN:=FALSE , PT:=T#50MS );
				iMainSetp:=300;
			ELSE
				 iMainSetp_TON[2](IN:=TRUE , PT:=T#50MS );
				 IF  iMainSetp_TON[2].Q THEN
					  iMainSetp_TON[2](IN:=FALSE , PT:=T#50MS );
					  iMainSetp:=400;   
				 END_IF
			 END_IF						
				
				
				
END_CASE

IF P3_SystemRUN.iMode=3 THEN
	P3_manual:=TRUE;
	ELSE
	P3_manual:=FALSE;	
	END_IF









(*
R_TRIG_Bt[1](CLK:= P3_SystemRUN.btnStart   OR  P3_SystemRUN.hmiStart  );
R_TRIG_Bt[2](CLK:= P3_SystemRUN.btnStop   OR  P3_SystemRUN.hmiStop);
R_TRIG_Bt[4](CLK:=   P3_SystemRUN.btnAuto OR  P3_SystemRUN.hmiAuto);
R_TRIG_Bt[5](CLK:=  NOT P3_SystemRUN.btnAuto);
R_TRIG_Bt[6](CLK:=P3_SystemRUN.btnEstop);
R_TRIG_Bt[7](CLK:=P3_SystemRUN.btnReset OR  P3_SystemRUN.hmiReset OR stSysState.hmiReset);
R_TRIG_Bt[8](CLK:=  NOT P3_SystemRUN.hmiAuto);

IF R_TRIG_Bt[4].Q THEN  //自动
	P3_SystemRUN.FlgAuto:=TRUE;
	P3_SystemRUN.FlgManua:=FALSE;
END_IF
IF R_TRIG_Bt[5].Q  OR  R_TRIG_Bt[8].Q   THEN  //手动
	P3_SystemRUN.FlgAuto:=FALSE;
	P3_SystemRUN.FlgManua:=TRUE;
END_IF
P3_SystemRUN.bReset:=R_TRIG_Bt[7].Q  OR  bInitReset    ;  //复位

IF NOT b_Alarm[4] THEN
	P3_SystemRUN.bAutoCondition:=TRUE;
ELSE	
P3_SystemRUN.bAutoCondition:=TRUE;
END_IF
//TON20(IN:=stSysState.btnReset AND stSysState.btnStop , PT:=T#5S , Q=> , ET=> ); //长按复位和停止5秒系统复位

CASE iMainSetp OF 
0://   INIT
    Init();
    P3_SystemRUN.iMode:=0;
 IF  P3_SystemRUN.bInitDone THEN
     iMainSetp:=88;	
  END_IF
88://切换手动
  IF  P3_SystemRUN.FlgManua THEN
	  iMainSetp:=300;
  END_IF
   
 (***********************手动*********************************) 
300:
   P3_SystemRUN.iMode:=3;
   iMainSetp:=350;  
   
350: 
  	IF  R_TRIG_Bt[1].Q  OR  P3_SystemRUN.hmiAuto THEN  //启动按钮  
		IF  P3_SystemRUN.FlgAuto  AND  P3_SystemRUN.bAutoCondition THEN //AND gstM1.IM1.bAutoCondition  暂时屏蔽
	      iMainSetp:=100;
	    END_IF
	END_IF 
	
	IF  P3_SystemRUN.FlgManua AND TON20.Q THEN  //系统清除
	   iMainSetp:=999;
	END_IF

 (************************自动********************************) 
100:
   P3_SystemRUN.iMode:=1;
   iMainSetp:=150;  
150:  //系统停止中......
    rtStoping(Clk:=P3_SystemRUN.FlgManua OR  P3_SystemRUN.btnStop   OR   P3_SystemRUN.bErrorStop );  //自动中触发手动 停止 按钮  stSysRun.bErrorStop 包括正极和负极
    IF rtStoping.Q AND NOT P3_SystemRUN.hmiAuto THEN //自动触发停止
		P3_SystemRUN.Stoping:=TRUE;
		iMainSetp:=160; //
	END_IF;
160: //判断停止完成
   (*	IF  P3_SystemRUN.bStopFinished  THEN
        P3_SystemRUN.bStopFinished :=FALSE;
        P3_SystemRUN.Stoping:=FALSE;
		iMainSetp:=300; 
	END_IF  ;*)
	iMainSetp:=300; 


 (************************急停********************************) 
400://Stoping
   P3_SystemRUN.iMode:=4;
    EStop();  
   iMainSetp:=450;  
      
450: //急停跳出 
	IF  NOT  P3_SystemRUN.btnEstop   THEN  
        tonEStop(IN:=FALSE , PT:=T#50MS );
	    iMainSetp:=0;
    ELSE
         tonEStop(IN:=TRUE , PT:=T#50MS );
         IF  tonEStop.Q THEN
              tonEStop(IN:=FALSE , PT:=T#50MS );
              iMainSetp:=400;   
         END_IF
   	 END_IF

END_CASE

IF P3_SystemRUN.hmiAuto THEN
	P3_SystemRUN.FlgManua:=FALSE;//叠台手动标志
	P3_SystemRUN.FlgAuto:=TRUE;//叠台自动标志
ELSE
	P3_SystemRUN.FlgManua:=TRUE;//叠台手动标志
	P3_SystemRUN.FlgAuto:=FALSE;//叠台自动标志	
END_IF

IF   P3_SystemRUN.btnEstop  AND  P3_SystemRUN.iMode<>4  THEN  //
	  iMainSetp:=400;
      P3_SystemRUN.bInitDone:=FALSE;
      P3_SystemRUN.bStopFinished :=FALSE;
      P3_SystemRUN.Stoping:=FALSE;
END_IF
*)


(***************程序调用*********************)

  // Auto1_Method();






    Condition();
    MotionBasic();
    CyBasic();
   
    TempBasic();
    Alarm();
    Pusle();
	
	//尾段
	LateBlanking_Alarm();
	LateBlanking_Auto1();
	LateBlanking_Auto2();
	LateBlanking_Auto3();
	LateBlanking_Auto4();
	LateBlanking_Auto5();
	LateBlanking_Auto6();
	LateBlanking_Auto7();
	LateBlanking_Auto8_01Sticke();
	LateBlanking_Auto9_02Sticke();
	LateBlanking_Auto1_Stick();
	LateBlanking_Condition();
	L_Init1();
	L_Init2();
	L_Init3();
	L_Init4();
	L_Init5();
	L_Init6();
	L_Init7();
	L_Init8();
	LateBlanking_Temperature();
	LateBlanking_Thickness_Test();
	LateBlanking_Weight_Test();
	LateBlankingCylinderManual();
	LateBlankingMotorManual();
	LateBlanking_Short_Test();
	LateBlanking_Scan();
	
	Output_statistics();
	MES_JT_ZT();
	LateBlanking_Tips();
	MQ_FSY();
	

//Auto();

ACTION Alarm:


(******************气缸报警*******************)
FOR K1:=1 TO MaxCy DO 
     arrCYOnAlarm[K1]:=  arrCyCtrl[K1] .Status.Error1;
     arrCYOFFAlarm[K1]:=  arrCyCtrl[K1] .Status.Error2;
END_FOR

bCYHaveAlarm:=FALSE;
FOR K1:=1 TO MaxCy DO 
      bCYHaveAlarm:=bCYHaveAlarm OR arrCYOnAlarm[K1] OR  arrCYOFFAlarm[K1];
END_FOR



(********轴报警**************)
FOR K1:=1 TO MaxAxes DO 
     arrAxisAlarm[K1]:=  arrAxis[K1] .Status.Error AND  arrAxis[K1] .Status.ErrorID<>16#42A0 ;
	 
END_FOR



bAxisHaveAlarm:=FALSE;
FOR K1:=1 TO MaxAxes DO 
      bAxisHaveAlarm:=bAxisHaveAlarm OR arrAxisAlarm[K1];
END_FOR




(*

(***超温报警*****自整定故障*****温控有报警*****)
FOR K1:=1 TO MaxTemp DO 
     arrTemHIAlarm[K1]:=         arrTempCtrl[K1].bTempError_HI ;
     arrTemSenserAlarm[K1]:=  arrTempCtrl[K1].bSenserError ;
     arrTemTuningAlarm[K1]:=  arrTempCtrl[K1].bTuningError ;
END_FOR

bTemHaveAlarm:=FALSE;
FOR K1:=1 TO MaxTemp DO 
      bTemHaveAlarm:=bTemHaveAlarm OR arrTemHIAlarm[K1]  OR   arrTemSenserAlarm[K1] OR   arrTemTuningAlarm[K1]  ;
END_FOR


(***************张力报警********************)
     arrTenAlarm[1]:=stP1PoleTen.bError;
     arrTenAlarm[2]:=stP1GMTen_U.bError;
     arrTenAlarm[3]:=stP1GMTen_D.bError;
     arrTenAlarm[4]:=stP1AuxDriverTen.bError;

     arrTenAlarm[5]:=stP2PoleTen_U.bError;
     arrTenAlarm[6]:=stP2PoleTen_D.bError;
     arrTenAlarm[7]:=stP2GMTen_U.bError;
     arrTenAlarm[8]:=stP2GMTen_D.bError;
     arrTenAlarm[9]:=stP2YFHTen.bError;

     arrTenAlarm[10]:=stP3PoleTen_U.bError;
     arrTenAlarm[11]:=stP3PoleTen_D.bError;

bTenHaveAlarm:=FALSE;
FOR K1:=1 TO 12 DO 
      bTenHaveAlarm:=bTenHaveAlarm OR arrTenAlarm[K1]   ;
END_FOR



(***************纠偏报警********************)
FOR K1:=1 TO MaxRec DO 
     arrRecAlarm[K1]:=arrRecCtrl[K1].Status.bError ;
END_FOR

bRecHaveAlarm:=FALSE;
FOR K1:=1 TO MaxRec DO 
      bRecHaveAlarm:=bRecHaveAlarm OR arrRecAlarm[K1]   ;
END_FOR



(***************创建凸轮报警*******************)
    arrCreatTableAlarm[1]:=stP1MQDriverCam.bCreatTableError;
    arrCreatTableAlarm[2]:=stP1MQCuterCam.bCreatTableError;
    arrCreatTableAlarm[3]:=stP1MQLineCam.bCreatTableError;
    arrCreatTableAlarm[4]:=stP1MQClampCam.bCreatTableError;
    arrCreatTableAlarm[5]:=stP1PoleBufferCam.bCreatTableError;

    arrCreatTableAlarm[6]:=stP2MQDriverCam_U.bCreatTableError;
    arrCreatTableAlarm[7]:=stP2MQCuterCam_U.bCreatTableError;
    arrCreatTableAlarm[8]:=stP2MQLineCam_U.bCreatTableError;
    arrCreatTableAlarm[9]:=stP2MQClampCam_U.bCreatTableError;
    arrCreatTableAlarm[10]:=stP2PoleBufferCam_U.bCreatTableError;

    arrCreatTableAlarm[11]:=stP2MQDriverCam_D.bCreatTableError;
    arrCreatTableAlarm[12]:=stP2MQCuterCam_D.bCreatTableError;
    arrCreatTableAlarm[13]:=stP2MQLineCam_D.bCreatTableError;
    arrCreatTableAlarm[14]:=stP2MQClampCam_D.bCreatTableError;
    arrCreatTableAlarm[15]:=stP2PoleBufferCam_D.bCreatTableError;

    arrCreatTableAlarm[16]:=stP3MQDriverCam_U.bCreatTableError;
    arrCreatTableAlarm[17]:=stP3MQCuterCam_U.bCreatTableError;
    arrCreatTableAlarm[18]:=stP3MQLineCam_U.bCreatTableError;
    arrCreatTableAlarm[19]:=stP3MQClampCam_U.bCreatTableError;
    arrCreatTableAlarm[20]:=stP3PoleBufferCam_U.bCreatTableError;

    arrCreatTableAlarm[21]:=stP3MQDriverCam_D.bCreatTableError;  
    arrCreatTableAlarm[22]:=stP3MQCuterCam_D.bCreatTableError;
    arrCreatTableAlarm[23]:=stP3MQLineCam_D.bCreatTableError;  
    arrCreatTableAlarm[24]:=stP3MQClampCam_D.bCreatTableError;
    arrCreatTableAlarm[25]:=stP3PoleBufferCam_D.bCreatTableError;  

  bCreatTableHaveAlarm:=FALSE;
  FOR K1:=1 TO 28 DO 
		bCreatTableHaveAlarm:=bCreatTableHaveAlarm OR arrCreatTableAlarm[K1]   ;
  END_FOR


(***************凸轮耦合报警*******************)
    arrCamInAlarm[1]:=stP1MQDriverCam.bError;
    arrCamInAlarm[2]:=stP1MQCuterCam.bError;
    arrCamInAlarm[3]:=stP1MQLineCam.bError;
    arrCamInAlarm[4]:=stP1MQClampCam.bError;
    arrCamInAlarm[5]:=stP1PoleBufferCam.bError;

    arrCamInAlarm[6]:=stP2MQDriverCam_U.bError;
    arrCamInAlarm[7]:=stP2MQCuterCam_U.bError;
    arrCamInAlarm[8]:=stP2MQLineCam_U.bError;
    arrCamInAlarm[9]:=stP2MQClampCam_U.bError;
    arrCamInAlarm[10]:=stP2PoleBufferCam_U.bError;

    arrCamInAlarm[11]:=stP2MQDriverCam_D.bError;
    arrCamInAlarm[12]:=stP2MQCuterCam_D.bError;
    arrCamInAlarm[13]:=stP2MQLineCam_D.bError;
    arrCamInAlarm[14]:=stP2MQClampCam_D.bError;
    arrCamInAlarm[15]:=stP2PoleBufferCam_D.bError;

    arrCamInAlarm[16]:=stP3MQDriverCam_U.bError;
    arrCamInAlarm[17]:=stP3MQCuterCam_U.bError;
    arrCamInAlarm[18]:=stP3MQLineCam_U.bError;
    arrCamInAlarm[19]:=stP3MQClampCam_U.bError;
    arrCamInAlarm[20]:=stP3PoleBufferCam_U.bError;

    arrCamInAlarm[21]:=stP3MQDriverCam_D.bError;  
    arrCamInAlarm[22]:=stP3MQCuterCam_D.bError;
    arrCamInAlarm[23]:=stP3MQLineCam_D.bError;  
    arrCamInAlarm[24]:=stP3MQClampCam_D.bError;
    arrCamInAlarm[25]:=stP3PoleBufferCam_D.bError;  
    arrCamInAlarm[26];  
  bCamHaveAlarm:=FALSE;
  FOR K1:=1 TO 28 DO 
		bCamHaveAlarm:=bCamHaveAlarm OR arrCamInAlarm[K1]   ;
  END_FOR


(***************齿轮报警*******************)
    arrGearAlarm[1]:=stP1YFHDriverGear_D.bError;
    arrGearAlarm[2]:=stP1YFHDriverInGear.bError;
    arrGearAlarm[3]:=stP1MQVirMainGear2.bError;

    arrGearAlarm[4]:=stP2GMDriverGear_D.bError;
    arrGearAlarm[5]:=stP2YFHDriverGear_U.bError;
    arrGearAlarm[6]:=stP2YFHDriverGear_D.bError;
    arrGearAlarm[7]:=stP2YFHDriverInGear.bError;
    arrGearAlarm[8]:=stP2MQVirMainGear_U.bError;
    arrGearAlarm[9]:=stP2MQVirMainGear_D.bError;

    arrGearAlarm[10]:=stP3YFHRollGear_U.bError;
    arrGearAlarm[11]:=stP3YFHRollGear_D.bError;
    arrGearAlarm[12]:=stP3YFHDriverGear_U.bError;
    arrGearAlarm[13]:=stP3YFHDriverGear_D.bError;
    arrGearAlarm[14]:=stP3YFHDriverInGear.bError;
    arrGearAlarm[15]:=stP3MQVirMainGear_U.bError;
    arrGearAlarm[16]:=stP3MQVirMainGear_D.bError;

    arrGearAlarm[17]:=stP1MQVirDriverGear.bError;
    arrGearAlarm[18]:=stP2MQVirDriverGear_U.bError;
    arrGearAlarm[19]:=stP2MQVirDriverGear_D.bError;
    arrGearAlarm[20]:=stP3MQVirDriverGear_U.bError;
     arrGearAlarm[21]:=stP3MQVirDriverGear_D.bError;


  bGearHaveAlarm:=FALSE;
  FOR K1:=1 TO 21 DO 
		bGearHaveAlarm:=bGearHaveAlarm OR arrGearAlarm[K1]   ;
  END_FOR




























(*

IF  iModeEN.bDoorEN THEN //屏蔽
   bDoor_Stop:=FALSE;
ELSE//屏蔽
  bDoor_Stop:=NOT stSysState.btnDoor[1] OR NOT stSysState.btnDoor[2] OR NOT stSysState.btnDoor[3] OR NOT stSysState.btnDoor[4] 
              OR NOT stSysState.btnDoor[5] OR NOT stSysState.btnDoor[6] OR NOT stSysState.btnDoor[7];
END_IF


bEstop:=stSysState.btnEstop[1] OR stSysState.btnEstop[2] OR stSysState.btnEstop[3] OR stSysState.btnEstop[4] OR stSysState.btnEstop[5];

(*===============================================报警信息============================================================*)
////判断是否有轴报警   arrError[1]
arrError[1]:=FALSE;
FOR I1:=1 TO MaxAxes BY 1 DO
	arrAxisError[I1] :=arrAxis[I1].Status.Error;  
    arrError[1]:= arrError[1] OR  arrAxisError[I1] ;	
END_FOR

(*****************M1 气缸报警****************) 
(*
arrActuatorsError[1]:= gstM1.acDriver1Press.Error;
arrActuatorsError[2]:= gstM1.acDriver2Press.Error;
arrActuatorsError[3]:= gstM1.acBoard1Press.Error;
arrActuatorsError[4]:= gstM1.acBoard2Press.Error ;

arrActuatorsError[11]:= gstM2.acPoleLock1.Error;
arrActuatorsError[12]:= gstM2.acPoleLock2.Error;
arrActuatorsError[13]:= gstM2.acBoxLock1.Error;
arrActuatorsError[14]:= gstM2.acBoxLock2.Error;
arrActuatorsError[15]:= gstM2.acDustClear1.Error ;
arrActuatorsError[16]:= gstM2.acDustClear2.Error ;
*)

(*****************功能报警****************)
arrFunctionError[1]:=gstM1.ctrlTension1.bError;
arrFunctionError[2]:=gstM1.ctrlTension2.bError;
arrFunctionError[3]:=gstM1.ctrlTension3.bError;
arrFunctionError[4]:=gstM1.ctrlTension4.bError;
arrFunctionError[5]:=gstM1.ctrlCuterCam.bError;
//arrFunctionError[6]:=gstM1.ctrlGearInVirDriver1.bError;
arrFunctionError[7]:=gstM1.ctrlRectify1.Error;
arrFunctionError[8]:=gstM1.ctrlRectify2.Error;

arrFunctionError[9]:=gstM2.ctrlGearBelt2.bError;
arrFunctionError[10]:=gstM2.ctrlVirBeltCan.bError;
arrFunctionError[11]:=gstM2.ctrlCcdCam.bError;
arrFunctionError[12]:=gstM2.ctrlNG1Cam.bError;
arrFunctionError[13]:=gstM2.ctrlNG2Cam.bError;
arrFunctionError[14]:=gstM2.ctrlOK1Cam.bError;
arrFunctionError[15]:=gstM2.ctrlOK2Cam.bError;

arrError[2]:=FALSE;
FOR I2:=1 TO 10 BY 1 DO  //红灯报警
    arrError[2]:= arrError[2] OR  arrActuatorsError[I2] ;	
END_FOR

arrError[3]:=FALSE;
FOR I5:=11 TO 20 BY 1 DO  //警告报警
    arrError[3]:= arrError[3] OR  arrActuatorsError[I5] ;	
END_FOR

arrError[4]:=FALSE;
FOR I4:=1 TO 20 BY 1 DO  //红灯报警
    arrError[4]:= arrError[4] OR  arrFunctionError[I4] ;	
END_FOR


stSysState.bAlarmStop:= arrError[1] OR arrError[2] OR arrError[4] ;


(*==============报警复位=========================*)
//轴  气缸报警  红灯亮       蜂鸣器 0.5秒 频率 响 8 秒后停止    

IF stSysState.iMode=3 THEN
	stSysState.bReset:=stSysState.btnReset;
END_IF

(*****蜂鸣器*****)
rt100(CLK:=arrError[1] OR arrError[2] OR arrError[4] , Q=> );
rt101(CLK:=arrError[3]  , Q=> );
IF rt100.Q THEN
	iErrorSetp:=100;//故障报警
END_IF

IF rt101.Q THEN
	iErrorSetp:=200;//警告报警
END_IF


tDelayBuzze(IN:= , PT:= , Q=> , ET=> );
CASE iErrorSetp   OF
100:
  tDelayBuzze.PT:=T#8S;
  tDelayBuzze.IN:=TRUE;
  iErrorSetp:=500;
200:
  tDelayBuzze.PT:=T#4S;
   tDelayBuzze.IN:=TRUE;
  iErrorSetp:=600;
500:
		stSysState.boBuzzer:= Pulse._250ms.Q;  //   (NOT bError1 AND NOT bError2) AND
		IF tDelayBuzze.Q  THEN
			iErrorSetp:=0;
			tDelayBuzze.IN:=FALSE;
			stSysState.boBuzzer:=FALSE;
		END_IF
600:
		stSysState.boBuzzer:= Pulse._1s.Q;  //    (NOT bError1 AND NOT bError2) AND
		IF tDelayBuzze.Q  THEN
			iErrorSetp:=0;
			tDelayBuzze.IN:=FALSE;
			stSysState.boBuzzer:=FALSE;
		END_IF

END_CASE


(*****三色灯控制*********)
//自动   绿
    RT200[1](CLK:=stSysState.iMode=1 , Q=> ); 
   IF RT200[1].Q THEN
	  bTurnOn:=TRUE;
      iLightSel:=3;
   END_IF       
//手动  黄
    RT200[2](CLK:=stSysState.iMode=3 , Q=> ); 
   IF RT200[2].Q THEN
	  bTurnOn:=TRUE;
      iLightSel:=2;
   END_IF 

//暂停   黄
    RT200[3](CLK:=stSysState.iMode=2 , Q=> ); 
   IF RT200[3].Q THEN
	  bTurnOn:=TRUE;
      iLightSel:=2;
   END_IF 
   
//暂停   红   //急停 OR 故障
    RT200[4](CLK:=stSysState.iMode=4  OR rt100.Q  , Q=> ); 
   IF RT200[4].Q THEN
	  bTurnOn:=TRUE;
      iLightSel:=1;
   END_IF    
   
IF bTurnOn THEN
	CASE iLightSel OF 
	  1: //红灯
		stSysState.boGreenLight:=FALSE;
		stSysState.boRedLight:=TRUE;
		stSysState.boYellowLight:=FALSE;
	
	  2://黄灯
		stSysState.boGreenLight:=FALSE;
		stSysState.boRedLight:=FALSE;
		stSysState.boYellowLight:=TRUE;
	
	  3://绿灯
		stSysState.boGreenLight:=TRUE;
		stSysState.boRedLight:=FALSE;
		stSysState.boYellowLight:=FALSE;
	
	END_CASE
   bTurnOn:=FALSE;
END_IF




*)
*)
END_ACTION

ACTION Condition:


IF arrAxisCtrlV2[P3AxisNo.P3_M2_OvenCarrying].Io.biNegLimit THEN    ////烤箱上料夹搬运电机
	 arrAxisCtrlV2[P3AxisNo.P3_M2_OvenCarrying].Cmd.JogN_Condition:=FALSE;
  ELSE
	 arrAxisCtrlV2[P3AxisNo.P3_M2_OvenCarrying].Cmd.JogN_Condition:=TRUE;
END_IF
IF arrAxisCtrlV2[P3AxisNo.P3_M2_OvenCarrying].Io.biPosLimit THEN
	 arrAxisCtrlV2[P3AxisNo.P3_M2_OvenCarrying].Cmd.JogP_Condition:=FALSE;
  ELSE
	 arrAxisCtrlV2[P3AxisNo.P3_M2_OvenCarrying].Cmd.JogP_Condition:=TRUE;
END_IF

IF arrAxisCtrlV2[P3AxisNo.P3_M2_OvenRetracting].Io.biNegLimit  THEN    ////烤箱上料夹进退电机
	 arrAxisCtrlV2[P3AxisNo.P3_M2_OvenRetracting].Cmd.JogN_Condition:=FALSE;
  ELSE
	 arrAxisCtrlV2[P3AxisNo.P3_M2_OvenRetracting].Cmd.JogN_Condition:=TRUE;
END_IF
IF arrAxisCtrlV2[P3AxisNo.P3_M2_OvenRetracting].Io.biPosLimit THEN
	 arrAxisCtrlV2[P3AxisNo.P3_M2_OvenRetracting].Cmd.JogP_Condition:=FALSE;
  ELSE
	 arrAxisCtrlV2[P3AxisNo.P3_M2_OvenRetracting].Cmd.JogP_Condition:=TRUE;
END_IF

IF arrAxisCtrlV2[P3AxisNo.P3_M2_OvenUpDown].Io.biNegLimit THEN    ////烤箱上料夹升降电机
	 arrAxisCtrlV2[P3AxisNo.P3_M2_OvenUpDown].Cmd.JogN_Condition:=FALSE;
  ELSE
	 arrAxisCtrlV2[P3AxisNo.P3_M2_OvenUpDown].Cmd.JogN_Condition:=TRUE;
END_IF
IF arrAxisCtrlV2[P3AxisNo.P3_M2_OvenUpDown].Io.biPosLimit THEN
	 arrAxisCtrlV2[P3AxisNo.P3_M2_OvenUpDown].Cmd.JogP_Condition:=FALSE;
  ELSE
	 arrAxisCtrlV2[P3AxisNo.P3_M2_OvenUpDown].Cmd.JogP_Condition:=TRUE;
END_IF







//MES下发数据写入
DT_To_MQ_MES.PostiveCode1:=P3_PLC_PC_MES.PostiveCode1;//正极左1条码		1
DT_To_MQ_MES.PostiveCode2:=P3_PLC_PC_MES.PostiveCode2;//正极右2条码		2
DT_To_MQ_MES.NegativeCode1:=P3_PLC_PC_MES.NegativeCode1;//负极左1条码		3
DT_To_MQ_MES.NegativeCode2:=P3_PLC_PC_MES.NegativeCode2;//负极右2条码		4
DT_To_MQ_MES.Station1_Code:=P3_PLC_PC_MES.Station1_Code;//叠台1隔膜条码		5
DT_To_MQ_MES.Station2_Code	:=P3_PLC_PC_MES.Station2_Code;//叠台2隔膜条码		6
DT_To_MQ_MES.Station3_Code	:=P3_PLC_PC_MES.Station3_Code;//叠台3隔膜条码		7
DT_To_MQ_MES.Station1_BlueCode:=P3_PLC_PC_MES.Station1_BlueCode;//叠台1l蓝胶条码		8
DT_To_MQ_MES.Station2_BlueCode:=P3_PLC_PC_MES.Station2_BlueCode;//叠台2蓝胶条码		9
DT_To_MQ_MES.Station3_BlueCode:=P3_PLC_PC_MES.Station3_BlueCode;//叠台3蓝胶条码		10
DT_To_MQ_MES.CellCode	:=P3_PLC_PC_MES.CellCode;//后段二维码胶条码	11
DT_To_MQ_MES.BlueCode:=P3_PLC_PC_MES.BlueCode;//后段蓝胶条码		12

//MES条码校验信号交互----PC_To_PLC
DT_To_MQ_MES.Mes_PcToPlc1:=P3_PLC_PC_MES. Mes_PcToPlc1       ;   //正极左1条码条码校验完成信号
DT_To_MQ_MES.Mes_PcToPlc2:=P3_PLC_PC_MES.Mes_PcToPlc2        ;   //正极右2条码校验完成信号
DT_To_MQ_MES.Mes_PcToPlc3:=P3_PLC_PC_MES.Mes_PcToPlc3        ;   //负极左1条码校验完成信号
DT_To_MQ_MES.Mes_PcToPlc4:=P3_PLC_PC_MES.Mes_PcToPlc4      ;   //负极右2条码校验完成信号
DT_To_MQ_MES.Mes_PcToPlc5:=P3_PLC_PC_MES.Mes_PcToPlc5      ;   //叠台1隔膜条码校验完成信号
DT_To_MQ_MES.Mes_PcToPlc6:=P3_PLC_PC_MES.Mes_PcToPlc6       ;   //叠台2隔膜条码校验完成信号
DT_To_MQ_MES.Mes_PcToPlc7:=P3_PLC_PC_MES.Mes_PcToPlc7       ;   //叠台3隔膜条码校验完成信号
DT_To_MQ_MES.Mes_PcToPlc8:=P3_PLC_PC_MES.Mes_PcToPlc8        ;   //叠台1l蓝胶条码校验完成信号
DT_To_MQ_MES.Mes_PcToPlc9:=P3_PLC_PC_MES.Mes_PcToPlc9       ;   //叠台2蓝胶条码校验完成信号
DT_To_MQ_MES.Mes_PcToPlc10:=P3_PLC_PC_MES.Mes_PcToPlc10        ;  //叠台3蓝胶条码校验完成信号
DT_To_MQ_MES.Mes_PcToPlc11:=P3_PLC_PC_MES.Mes_PcToPlc11      ;   //后段二维码胶条码校验完成信号
DT_To_MQ_MES.Mes_PcToPlc12:=P3_PLC_PC_MES.Mes_PcToPlc12       ;   //后段蓝胶条码校验完成信号	




//MES物料码交互------------条码清理及校验完成信号清理
//正极
rMES[1](CLK:=MQ_To_DT_MES.Mes_PlcToPc1,Q=>);
rMES[2](CLK:=MQ_To_DT_MES.Mes_PlcToPc2,Q=>);
rMES[3](CLK:=MQ_To_DT_MES.Mes_PlcToPc3,Q=>);
rMES[4](CLK:=MQ_To_DT_MES.Mes_PlcToPc4,Q=>);

IF rMES[1].Q THEN//正极左换卷---请求换卷时清当前条码
	P3_PLC_PC_MES.PostiveCode1:='';
	P3_PLC_PC_MES.Mes_PcToPlc1:=FALSE;
	DT_To_MQ_MES.MesClear_Pc1:=TRUE;
END_IF
IF rMES[2].Q THEN//正极右换卷---请求换卷时清当前条码
	P3_PLC_PC_MES.PostiveCode2:='';
	P3_PLC_PC_MES.Mes_PcToPlc2:=FALSE;
	DT_To_MQ_MES.MesClear_Pc2:=TRUE;
END_IF
//负极
IF rMES[3].Q THEN//负极左换卷---请求换卷时清当前条码
	P3_PLC_PC_MES.NegativeCode1:='';
	P3_PLC_PC_MES.Mes_PcToPlc3:=FALSE;
	DT_To_MQ_MES.MesClear_Pc3:=TRUE;
END_IF
IF rMES[4].Q THEN//负极右换卷---请求换卷时清当前条码
	P3_PLC_PC_MES.NegativeCode2:='';
	P3_PLC_PC_MES.Mes_PcToPlc4:=FALSE;
	DT_To_MQ_MES.MesClear_Pc4:=TRUE;
END_IF

tMES[1](IN:=DT_To_MQ_MES.MesClear_Pc1 , PT:=T#100MS , Q=> , ET=> );
tMES[2](IN:=DT_To_MQ_MES.MesClear_Pc2 , PT:=T#100MS , Q=> , ET=> );
tMES[3](IN:=DT_To_MQ_MES.MesClear_Pc3 , PT:=T#100MS , Q=> , ET=> );
tMES[4](IN:=DT_To_MQ_MES.MesClear_Pc4 , PT:=T#100MS , Q=> , ET=> );
IF tMES[1].Q THEN
	DT_To_MQ_MES.MesClear_Pc1:=FALSE;
END_IF
IF tMES[2].Q THEN
	DT_To_MQ_MES.MesClear_Pc2:=FALSE;
END_IF
IF tMES[3].Q THEN
	DT_To_MQ_MES.MesClear_Pc3:=FALSE;
END_IF
IF tMES[4].Q THEN
	DT_To_MQ_MES.MesClear_Pc4:=FALSE;
END_IF






//后段二维码条码校验
IF  (P3_PLC_PC_MES.Mes_PcToPlc11 AND  LEN(P3_PLC_PC_MES.CellCode)>6  ) OR P3User2_Par.Shield[8] THEN
	StickIDGlue.IDGlueNumberOK:=TRUE;
ELSE
	StickIDGlue.IDGlueNumberOK:=FALSE;
END_IF

IF StickIDGlue.IDGlueNumberOK THEN//二维码料号OK
	CellMemory[12].P3CellCode :=P3_PLC_PC_MES.CellCode;	
ELSE
	CellMemory[12].P3CellCode :='';	
END_IF
//二维码条码重新校验

rMES[5](CLK:=P3User2_Par.Shield[9] , Q=> );  //二维码胶有无料检测报警
IF rMES[5].Q THEN
	StickIDGlue.IDGlueNumberOK:=FALSE;
	P3_PLC_PC_MES.CellCode:='';
	P3_PLC_PC_MES.Mes_PcToPlc11:=FALSE;
END_IF	


//后段蓝胶重新校验
IF  (P3_PLC_PC_MES.Mes_PcToPlc12 AND  LEN(P3_PLC_PC_MES.BlueCode)>6  ) OR P3User2_Par.Shield[8] THEN
	BlueGlueNumberOK:=TRUE;//蓝胶条码校验OK
ELSE
	BlueGlueNumberOK:=FALSE;//蓝胶条码校验OK
END_IF

IF BlueGlueNumberOK THEN//蓝胶条码
	CellMemory[12].P3BlueCode :=P3_PLC_PC_MES.BlueCode;	
ELSE
	CellMemory[12].P3BlueCode :='';	
END_IF
//蓝胶条码重新校验
rMES[6](CLK:=P3User2_Par.Shield[10] , Q=> );   //蓝胶有无料检测报警
IF rMES[6].Q THEN
	BlueGlueNumberOK:=FALSE;
	P3_PLC_PC_MES.BlueCode:='';
	P3_PLC_PC_MES.Mes_PcToPlc12:=FALSE;
END_IF	


IF NOT  StickIDGlue.IDGlueNumberOK AND NOT P3User2_Par.Shield[8] THEN
	P3_Error[57]:=TRUE;//后段二维码条码校验未通过
ELSE
	P3_Error[57]:=FALSE;//后段二维码条码校验未通过
END_IF
IF NOT  BlueGlueNumberOK AND NOT P3User2_Par.Shield[8] THEN
	P3_Error[58]:=TRUE;//后段蓝胶条码校验未通过
ELSE
	P3_Error[58]:=FALSE;//后段蓝胶条码校验未通过
END_IF



(*
PostiveCode1				:STRING;//正极左1条码		1
PostiveCode2				:STRING;//正极右2条码		2
NegativeCode1				:STRING;//负极左1条码		3
NegativeCode2				:STRING;//负极右2条码		4
Station1_Code				:STRING;//叠台1隔膜条码		5
Station2_Code				:STRING;//叠台2隔膜条码		6
Station3_Code				:STRING;//叠台3隔膜条码		7
Station1_BlueCode			:STRING;//叠台1l蓝胶条码		8
Station2_BlueCode			:STRING;//叠台2蓝胶条码		9
Station3_BlueCode			:STRING;//叠台3蓝胶条码		10
CellCode					:STRING;//后段二维码胶条码	11
BlueCode					:STRING;//后段蓝胶条码		12

//MES条码校验信号交互----PC_To_PLC
Mes_PcToPlc1:        BOOL;   //正极左1条码条码校验完成信号
Mes_PcToPlc2:        BOOL;   //正极右2条码校验完成信号
Mes_PcToPlc3:        BOOL;   //负极左1条码	校验完成信号
Mes_PcToPlc4:        BOOL;   //负极右2条码校验完成信号
Mes_PcToPlc5:        BOOL;   //叠台1隔膜条码校验完成信号
Mes_PcToPlc6:        BOOL;   //叠台2隔膜条码校验完成信号
Mes_PcToPlc7:        BOOL;   //叠台3隔膜条码校验完成信号
Mes_PcToPlc8:        BOOL;   //叠台1l蓝胶条码校验完成信号
Mes_PcToPlc9:        BOOL;   //叠台2蓝胶条码校验完成信号
Mes_PcToPlc10:        BOOL;  //叠台3蓝胶条码校验完成信号
Mes_PcToPlc11:        BOOL;   //后段二维码胶条码校验完成信号
Mes_PcToPlc12:        BOOL;   //后段蓝胶条码校验完成信号	

*)
END_ACTION

ACTION CyBasic:

//气缸控制   刷新周期可以慢
FOR i:=230 TO 289  DO//MaxCy
	  fbCy[i](bReset:=P3_SystemRUN.bReset ,AutoRun:=P3_SystemRUN.iMode=1 , stCyCtrl:=arrCyCtrl[i] );
    //fbCy[i](bReset:=P3_SystemRUN.bReset , stCyCtrl:=arrCyCtrl[i] );
END_FOR
END_ACTION

ACTION EStop:

//CASE iMainEStopSetp OF




 FOR I1:=160 TO 185 BY 1 DO//MaxAxes
	IF I1<=165 OR I1>=169 THEN
		arrAxisCtrl[I1].Cmd. bHome:=FALSE;
		arrAxisCtrl[I1].Cmd. bJog_Bw:=FALSE;	
		arrAxisCtrl[I1].Cmd. bJog_Fw:=FALSE;		
		arrAxisCtrl[I1].Cmd. bMoveAbs:=FALSE;		
		arrAxisCtrl[I1].Cmd. bMoveRel:=FALSE;	
		arrAxisCtrl[I1].Cmd. bMoveVelo:=FALSE;		
		arrAxisCtrl[I1].Cmd.bMoveModulo:=FALSE;	
		arrAxisCtrl[I1].Cmd. bSetPos:=FALSE;	    	
		arrAxisCtrl[I1].Cmd. iGoSetPos:=0;	  		
		//arrAxisCtrl[I1].bEnable:=TRUE;
		IF  arrAxisCtrl[I1].Status.Moving  AND NOT arrAxisCtrl[I1].Cmd.bStop   AND  NOT arrAxis[I1] .Status.Coupled THEN   //对运动中的轴执行STOP
	    	arrAxisCtrl[I1].Cmd. bStop:=TRUE;	
		END_IF;		
   END_IF 
   IF I1>=166 AND I1<=168 THEN
		arrAxisCtrlV2[I1].Cmd. bHome:=FALSE;
		arrAxisCtrlV2[I1].Cmd. bJog_Bw:=FALSE;	
		arrAxisCtrlV2[I1].Cmd. bJog_Fw:=FALSE;		
		arrAxisCtrlV2[I1].Cmd. bMoveAbs:=FALSE;		
		arrAxisCtrlV2[I1].Cmd. bMoveRel:=FALSE;	
		arrAxisCtrlV2[I1].Cmd. bMoveVelo:=FALSE;		
		arrAxisCtrlV2[I1].Cmd.bMoveModulo:=FALSE;	
		arrAxisCtrlV2[I1].Cmd. bSetPos:=FALSE;	    	
		arrAxisCtrlV2[I1].Cmd. iGoSetPos:=0;	  		
//arrAxisCtrl[I1].bEnable:=TRUE;
IF  arrAxisCtrlV2[I1].Status.Moving  AND NOT arrAxisCtrlV2[I1].Cmd.bStop   AND  NOT arrAxis[I1] .Status.Coupled THEN   //对运动中的轴执行STOP
arrAxisCtrl[I1].Cmd. bStop:=TRUE;	
		END_IF;		
   END_IF
  END_FOR;
END_ACTION

ACTION Init:

//整机初始化
(**
1.P1INIT  
2.P2INIT
3.P3INIT
4.P4INIT
5.缓存凸轮表创建
6.Time轴跑速度模式
*)

CASE iMainInitSetp OF
0:
    IF  NOT   P3_SystemRUN.bInitDone THEN
         iMainInitSetp:=10;
    END_IF
10:
    FOR i:=160 TO 185  DO 
		IF i<=165 OR i>=169 THEN
			arrAxisCtrl[i].Cmd.bEnable:=TRUE;
			arrAxisCtrl[i].Cmd.bEnableFw:=TRUE;
			arrAxisCtrl[i].Cmd.bEnableBw:=TRUE;
			(*其他操作指令*)  
			arrAxisCtrl[i].Cmd.bHome:=FALSE;
			arrAxisCtrl[i].Cmd.bJog_Bw:=FALSE;
			arrAxisCtrl[i].Cmd.bHalt:=FALSE;
			arrAxisCtrl[i].Cmd.bJog_Fw:=FALSE;
			arrAxisCtrl[i].Cmd.bMoveAbs:=FALSE;
			arrAxisCtrl[i].Cmd.bMoveVelo:=FALSE;
			arrAxisCtrl[i].Cmd.bMoveRel:=FALSE;
			arrAxisCtrl[i].Cmd.bReset:=FALSE;
			arrAxisCtrl[i].Cmd.bStop:=FALSE;
			arrAxisCtrl[i].Cmd.bSetPos:=FALSE;
			arrAxisPar[i].bLimitSwitchEn:=TRUE;
		
		
			arrAxisCtrl[i].Cmd.Home_Condition:=TRUE;
			arrAxisCtrl[i].Cmd.JogN_Condition:=TRUE;
			arrAxisCtrl[i].Cmd.JogP_Condition:=TRUE;		
		END_IF
		
		IF i>=166 AND i<=168 THEN
			arrAxisCtrlV2[i].Cmd.bEnable:=TRUE;
			arrAxisCtrlV2[i].Cmd.bEnableFw:=TRUE;
			arrAxisCtrlV2[i].Cmd.bEnableBw:=TRUE;
			(*其他操作指令*)  
			arrAxisCtrlV2[i].Cmd.bHome:=FALSE;
			arrAxisCtrlV2[i].Cmd.bJog_Bw:=FALSE;
			arrAxisCtrlV2[i].Cmd.bHalt:=FALSE;
			arrAxisCtrlV2[i].Cmd.bJog_Fw:=FALSE;
			arrAxisCtrlV2[i].Cmd.bMoveAbs:=FALSE;
			arrAxisCtrlV2[i].Cmd.bMoveVelo:=FALSE;
			arrAxisCtrlV2[i].Cmd.bMoveRel:=FALSE;
			arrAxisCtrlV2[i].Cmd.bReset:=FALSE;
			arrAxisCtrlV2[i].Cmd.bStop:=FALSE;
			arrAxisCtrlV2[i].Cmd.bSetPos:=FALSE;
			
		
			arrAxisCtrlV2[i].Cmd.Home_Condition:=TRUE;
			arrAxisCtrlV2[i].Cmd.JogN_Condition:=TRUE;
			arrAxisCtrlV2[i].Cmd.JogP_Condition:=TRUE;			
		END_IF
    END_FOR
    
    K1:=0;
    iMainInitSetp:=20;
20: //复位一次
   bInitReset:=TRUE;
   iMainInitSetp:=30;
30:
   K1:=K1+1;
   IF  K1>=10 THEN
        bInitReset:=FALSE;
        iMainInitSetp:=40;
   ELSE
     iMainInitSetp:=20;
   END_IF

40://P1---P4 Init
  P3_SystemRUN.bInitDone:=TRUE;
  P3_SystemRUN.TheFirstTimebool:=TRUE;
  iMainInitSetp:=0;
END_CASE
END_ACTION

ACTION MotionBasic:

FOR i:=160 TO MaxP3Axes DO
	IF i<=165 OR i>=169 THEN
  		csAxis[i](bReset:=P3_SystemRUN.bReset ,AutoRun:=P3_SystemRUN.iMode=1, Axis:=arrAxis[i] , stAxisCtrl:=arrAxisCtrl[i] , stAxisPar:=arrAxisPar[i] );
 	 END_IF
	 IF i>=166 AND i<=168 THEN
		csAxisV2[i](bReset:=P3_SystemRUN.bReset , AutoRun:=P3_SystemRUN.iMode=1,Axis:=arrAxis[i] , stAxisCtrl:=arrAxisCtrlV2[i] , stAxisPar:=arrAxisParV2[i] ); 
	 END_IF
END_FOR
(*
//		
FOR i:=160 TO MaxP3Axes DO
	IF i<=165 OR i>=169 THEN
  		csAxis[i](bReset:=P3_SystemRUN.bReset , Axis:=arrAxis[i] , stAxisCtrl:=arrAxisCtrl[i] , stAxisPar:=arrAxisPar[i] );
 	 END_IF
	 IF i>=166 AND i<=168 THEN
		csAxisV2[i](bReset:=P3_SystemRUN.bReset , Axis:=arrAxis[i] , stAxisCtrl:=arrAxisCtrlV2[i] , stAxisPar:=arrAxisParV2[i] ); 
	 END_IF
END_FOR

*)





(*
fbP4NGSetpMoter(stSetpMotor:=stP4NgPushMoter );//P4NG 排杆电机

fbP4CutElectric_CY(
	bServON:=               stP4CutCtrl.bServON , 
	bHome:=                  stP4CutCtrl.bHome , 
	bReset:=                   stSysState.bReset , 
	bStop:=                    stP4CutCtrl.bStop , 
	bJog_P:=                   stP4CutCtrl.bJog_P, 
	bJog_N:=                   stP4CutCtrl.bJog_N, 
	Pos_Start:=                 stP4CutCtrl.Pos_Start, 
	fTagetPos:=               stP4CutCtrl.fTagetPos , 
	fVel:=                       500  , //stP4CutCtrl.fVel
	fAcc:=                       8000 , //  stP4CutCtrl.fAcc
	fDec:=                      8000 , //stP4CutCtrl.fDec
	Delay_Time:=             T#5S , 
	bHomed=>               stP4CutCtrl.bHomed  , 
	Pos_Done=>             stP4CutCtrl.Pos_Done, 
	Home_Alm=>            stP4CutCtrl.Home_Alm, 
	Pos_Alm=>                stP4CutCtrl.Pos_Alm , 
	stJXCE:=                    stP4Cut                    );
stP4Cut.in_Act_Pos;


//stP4CutCtrl.bStop:=(stP4CutCtrl.Home_Alm OR   stP4CutCtrl.Pos_Alm ) AND stSysState.bReset;


IF stSysState.bReset THEN
  IF  arrAxis[VirAxisNo.P2_VirTimeWind].Status.ControlLoopClosed  AND arrAxis[VirAxisNo.P2_VirTimeWind].Status.NotMoving   THEN
	  arrAxisPar[VirAxisNo.P2_VirTimeWind].fVelocity_of_Velo:=100;
	  arrAxisCtrl[VirAxisNo.P2_VirTimeWind].Cmd.bMoveVelo:=TRUE;
  END_IF
END_IF

mc_Home(
	Axis:=                    arrAxis[71]  , 
	Execute:=              Execute , 
	Position:=            66 , 
	HomingMode:=  Tc2_MC2.MC_Direct , 
	BufferMode:= , 
	Options:= , 
	bCalibrationCam:=TRUE , 
	Done=> , 
	Busy=> , 
	Active=> , 
	CommandAborted=> , 
	Error=> , 
	ErrorID=> );


mc_Home.Done;
mc_Home.Busy;


fbCoeWrite_GlueFeed(
	sNetId:='192.168.20.10.6.1' , 
	nSlaveAddr:=  1015, 
	nSubIndex:=    16#1F, 
	nIndex:=        16#2005, 
	pSrcBuf:=ADR(wEncodeHome) , 
	cbBufLen:= 2, 
	bExecute:=bCoeWrite_GlueFeed , 
	tTimeout:= , 
	bBusy=> , 
	bError=> , 
	nErrId=> );





*)
END_ACTION

ACTION Pusle:
(*
/////////////////////////////////////////时钟脉冲////////////////////////////////////////////////////////////
//fbPulseCtrl1(PT_OFF:=T#2MS, PT_ON:=T#2MS, Q=>, RT=>);
fbPulseCtrl[1](PT_OFF:=T#2MS, PT_ON:=T#2MS,   );
fbPulseCtrl[2](PT_OFF:=T#4MS, PT_ON:=T#4MS,    );
fbPulseCtrl[3](PT_OFF:=T#10MS, PT_ON:=T#10MS,   );

fbPulseCtrl[4](PT_OFF:=T#300MS, PT_ON:=T#300MS,   );
fbPulseCtrl[5](PT_OFF:=T#3S, PT_ON:=T#3S,    );
fbPulseCtrl[6](PT_OFF:=T#5S, PT_ON:=T#5S,   );
fbPulseCtrl[7](PT_OFF:=T#10S, PT_ON:=T#10S,  );
fbPulseCtrl[8](PT_OFF:=T#250MS, PT_ON:=T#250MS,   );

fbPulseCtrl[9](PT_OFF:=T#2S, PT_ON:=T#200MS,   );

